LIN {X 98.094,Y 103.990,Z 85.740,A 180.000,B 0.000,C 180.000} C_DIS
LIN {X 98.166,Y 103.986,Z 85.738,A 180.000,B 0.000,C 180.000} C_DIS
LIN {X 98.239,Y 103.980,Z 85.735,A 180.000,B 0.000,C 180.000} C_DIS
LIN {X 98.312,Y 103.973,Z 85.733,A 180.000,B 0.000,C 180.000} C_DIS
LIN {X 98.387,Y 103.963,Z 85.730,A 180.000,B 0.000,C 180.000} C_DIS
LIN {X 98.462,Y 103.954,Z 85.727,A 180.000,B 0.000,C 180.000} C_DIS
LIN {X 98.537,Y 103.942,Z 85.725,A 180.000,B 0.000,C 180.000} C_DIS
LIN {X 98.612,Y 103.930,Z 85.722,A 180.000,B 0.000,C 180.000} C_DIS
LIN {X 98.763,Y 103.903,Z 85.717,A 180.000,B 0.000,C 180.000} C_DIS
LIN {X 98.839,Y 103.890,Z 85.714,A 180.000,B 0.000,C 180.000} C_DIS
LIN {X 98.915,Y 103.876,Z 85.711,A 180.000,B 0.000,C 180.000} C_DIS
LIN {X 98.986,Y 103.863,Z 85.709,A 180.000,B 0.000,C 180.000} C_DIS
LIN {X 99.057,Y 103.847,Z 85.706,A 180.000,B 0.000,C 180.000} C_DIS
LIN {X 99.128,Y 103.830,Z 85.704,A 180.000,B 0.000,C 180.000} C_DIS
LIN {X 99.199,Y 103.813,Z 85.701,A 180.000,B 0.000,C 180.000} C_DIS
LIN {X 99.271,Y 103.794,Z 85.699,A 180.000,B 0.000,C 180.000} C_DIS
LIN {X 99.343,Y 103.773,Z 85.696,A 180.000,B 0.000,C 180.000} C_DIS
LIN {X 99.415,Y 103.751,Z 85.693,A 180.000,B 0.000,C 180.000} C_DIS
LIN {X 99.487,Y 103.729,Z 85.691,A 180.000,B 0.000,C 180.000} C_DIS
LIN {X 99.634,Y 103.684,Z 85.685,A 180.000,B 0.000,C 180.000} C_DIS
LIN {X 99.708,Y 103.661,Z 85.683,A 180.000,B 0.000,C 180.000} C_DIS
LIN {X 99.781,Y 103.637,Z 85.680,A 180.000,B 0.000,C 180.000} C_DIS
LIN {X 99.849,Y 103.613,Z 85.677,A 180.000,B 0.000,C 180.000} C_DIS
LIN {X 99.917,Y 103.588,Z 85.675,A 180.000,B 0.000,C 180.000} C_DIS
LIN {X 99.985,Y 103.562,Z 85.672,A 180.000,B 0.000,C 180.000} C_DIS
LIN {X 100.052,Y 103.534,Z 85.670,A 180.000,B 0.000,C 180.000} C_DIS
LIN {X 100.122,Y 103.504,Z 85.667,A 180.000,B 0.000,C 180.000} C_DIS
LIN {X 100.193,Y 103.473,Z 85.665,A 180.000,B 0.000,C 180.000} C_DIS
LIN {X 100.402,Y 103.379,Z 85.657,A 180.000,B 0.000,C 180.000} C_DIS
LIN {X 100.471,Y 103.347,Z 85.654,A 180.000,B 0.000,C 180.000} C_DIS
LIN {X 100.539,Y 103.314,Z 85.651,A 180.000,B 0.000,C 180.000} C_DIS
LIN {X 100.607,Y 103.280,Z 85.649,A 180.000,B 0.000,C 180.000} C_DIS
LIN {X 100.672,Y 103.247,Z 85.646,A 180.000,B 0.000,C 180.000} C_DIS
LIN {X 100.735,Y 103.212,Z 85.643,A 180.000,B 0.000,C 180.000} C_DIS
LIN {X 100.799,Y 103.176,Z 85.641,A 180.000,B 0.000,C 180.000} C_DIS
LIN {X 100.862,Y 103.139,Z 85.638,A 180.000,B 0.000,C 180.000} C_DIS
LIN {X 100.929,Y 103.099,Z 85.636,A 180.000,B 0.000,C 180.000} C_DIS
LIN {X 101.127,Y 102.977,Z 85.628,A 180.000,B 0.000,C 180.000} C_DIS
LIN {X 101.190,Y 102.938,Z 85.625,A 180.000,B 0.000,C 180.000} C_DIS
LIN {X 101.253,Y 102.897,Z 85.622,A 180.000,B 0.000,C 180.000} C_DIS
LIN {X 101.315,Y 102.856,Z 85.620,A 180.000,B 0.000,C 180.000} C_DIS
LIN {X 101.376,Y 102.813,Z 85.617,A 180.000,B 0.000,C 180.000} C_DIS
LIN {X 101.437,Y 102.769,Z 85.615,A 180.000,B 0.000,C 180.000} C_DIS
LIN {X 101.497,Y 102.725,Z 85.612,A 180.000,B 0.000,C 180.000} C_DIS
LIN {X 101.556,Y 102.680,Z 85.609,A 180.000,B 0.000,C 180.000} C_DIS
LIN {X 101.614,Y 102.633,Z 85.607,A 180.000,B 0.000,C 180.000} C_DIS
LIN {X 101.736,Y 102.536,Z 85.601,A 180.000,B 0.000,C 180.000} C_DIS
LIN {X 101.797,Y 102.487,Z 85.599,A 180.000,B 0.000,C 180.000} C_DIS
LIN {X 101.858,Y 102.437,Z 85.596,A 180.000,B 0.000,C 180.000} C_DIS
LIN {X 101.914,Y 102.391,Z 85.593,A 180.000,B 0.000,C 180.000} C_DIS
LIN {X 101.969,Y 102.343,Z 85.591,A 180.000,B 0.000,C 180.000} C_DIS
LIN {X 102.023,Y 102.293,Z 85.588,A 180.000,B 0.000,C 180.000} C_DIS
LIN {X 102.077,Y 102.244,Z 85.586,A 180.000,B 0.000,C 180.000} C_DIS
LIN {X 102.132,Y 102.191,Z 85.583,A 180.000,B 0.000,C 180.000} C_DIS
LIN {X 102.186,Y 102.137,Z 85.580,A 180.000,B 0.000,C 180.000} C_DIS
LIN {X 102.239,Y 102.082,Z 85.578,A 180.000,B 0.000,C 180.000} C_DIS
LIN {X 102.292,Y 102.027,Z 85.575,A 180.000,B 0.000,C 180.000} C_DIS
LIN {X 102.399,Y 101.917,Z 85.570,A 180.000,B 0.000,C 180.000} C_DIS
LIN {X 102.452,Y 101.862,Z 85.567,A 180.000,B 0.000,C 180.000} C_DIS
LIN {X 102.504,Y 101.806,Z 85.564,A 180.000,B 0.000,C 180.000} C_DIS
LIN {X 102.553,Y 101.749,Z 85.562,A 180.000,B 0.000,C 180.000} C_DIS
LIN {X 102.603,Y 101.692,Z 85.559,A 180.000,B 0.000,C 180.000} C_DIS
LIN {X 102.651,Y 101.635,Z 85.556,A 180.000,B 0.000,C 180.000} C_DIS
LIN {X 102.698,Y 101.575,Z 85.554,A 180.000,B 0.000,C 180.000} C_DIS
LIN {X 102.745,Y 101.515,Z 85.551,A 180.000,B 0.000,C 180.000} C_DIS
LIN {X 102.791,Y 101.455,Z 85.548,A 180.000,B 0.000,C 180.000} C_DIS
LIN {X 102.929,Y 101.272,Z 85.540,A 180.000,B 0.000,C 180.000} C_DIS
LIN {X 102.974,Y 101.211,Z 85.538,A 180.000,B 0.000,C 180.000} C_DIS
LIN {X 103.018,Y 101.148,Z 85.535,A 180.000,B 0.000,C 180.000} C_DIS
LIN {X 103.061,Y 101.085,Z 85.532,A 180.000,B 0.000,C 180.000} C_DIS
LIN {X 103.102,Y 101.024,Z 85.530,A 180.000,B 0.000,C 180.000} C_DIS
LIN {X 103.141,Y 100.961,Z 85.527,A 180.000,B 0.000,C 180.000} C_DIS
LIN {X 103.180,Y 100.898,Z 85.525,A 180.000,B 0.000,C 180.000} C_DIS
LIN {X 103.218,Y 100.835,Z 85.522,A 180.000,B 0.000,C 180.000} C_DIS
LIN {X 103.257,Y 100.767,Z 85.519,A 180.000,B 0.000,C 180.000} C_DIS
LIN {X 103.335,Y 100.632,Z 85.514,A 180.000,B 0.000,C 180.000} C_DIS
LIN {X 103.373,Y 100.564,Z 85.511,A 180.000,B 0.000,C 180.000} C_DIS
LIN {X 103.409,Y 100.498,Z 85.509,A 180.000,B 0.000,C 180.000} C_DIS
LIN {X 103.444,Y 100.433,Z 85.506,A 180.000,B 0.000,C 180.000} C_DIS
LIN {X 103.479,Y 100.367,Z 85.503,A 180.000,B 0.000,C 180.000} C_DIS
LIN {X 103.511,Y 100.300,Z 85.501,A 180.000,B 0.000,C 180.000} C_DIS
LIN {X 103.543,Y 100.231,Z 85.498,A 180.000,B 0.000,C 180.000} C_DIS
LIN {X 103.575,Y 100.162,Z 85.495,A 180.000,B 0.000,C 180.000} C_DIS
LIN {X 103.605,Y 100.093,Z 85.493,A 180.000,B 0.000,C 180.000} C_DIS
LIN {X 103.694,Y 99.878,Z 85.485,A 180.000,B 0.000,C 180.000} C_DIS
LIN {X 103.724,Y 99.806,Z 85.482,A 180.000,B 0.000,C 180.000} C_DIS
LIN {X 103.753,Y 99.734,Z 85.479,A 180.000,B 0.000,C 180.000} C_DIS
LIN {X 103.780,Y 99.664,Z 85.477,A 180.000,B 0.000,C 180.000} C_DIS
LIN {X 103.805,Y 99.594,Z 85.474,A 180.000,B 0.000,C 180.000} C_DIS
LIN {X 103.829,Y 99.524,Z 85.471,A 180.000,B 0.000,C 180.000} C_DIS
LIN {X 103.853,Y 99.453,Z 85.469,A 180.000,B 0.000,C 180.000} C_DIS
LIN {X 103.875,Y 99.380,Z 85.466,A 180.000,B 0.000,C 180.000} C_DIS
LIN {X 103.896,Y 99.306,Z 85.463,A 180.000,B 0.000,C 180.000} C_DIS
LIN {X 103.916,Y 99.232,Z 85.461,A 180.000,B 0.000,C 180.000} C_DIS
LIN {X 103.978,Y 99.008,Z 85.453,A 180.000,B 0.000,C 180.000} C_DIS
LIN {X 103.998,Y 98.933,Z 85.450,A 180.000,B 0.000,C 180.000} C_DIS
LIN {X 104.016,Y 98.858,Z 85.447,A 180.000,B 0.000,C 180.000} C_DIS
LIN {X 104.032,Y 98.785,Z 85.445,A 180.000,B 0.000,C 180.000} C_DIS
LIN {X 104.047,Y 98.712,Z 85.442,A 180.000,B 0.000,C 180.000} C_DIS
LIN {X 104.062,Y 98.639,Z 85.439,A 180.000,B 0.000,C 180.000} C_DIS
LIN {X 104.074,Y 98.565,Z 85.437,A 180.000,B 0.000,C 180.000} C_DIS
LIN {X 104.086,Y 98.489,Z 85.434,A 180.000,B 0.000,C 180.000} C_DIS
LIN {X 104.097,Y 98.412,Z 85.431,A 180.000,B 0.000,C 180.000} C_DIS
LIN {X 104.130,Y 98.183,Z 85.423,A 180.000,B 0.000,C 180.000} C_DIS
LIN {X 104.140,Y 98.107,Z 85.421,A 180.000,B 0.000,C 180.000} C_DIS
LIN {X 104.148,Y 98.032,Z 85.418,A 180.000,B 0.000,C 180.000} C_DIS
LIN {X 104.155,Y 97.956,Z 85.415,A 180.000,B 0.000,C 180.000} C_DIS
LIN {X 104.162,Y 97.880,Z 85.413,A 180.000,B 0.000,C 180.000} C_DIS
LIN {X 104.166,Y 97.803,Z 85.410,A 180.000,B 0.000,C 180.000} C_DIS
LIN {X 104.169,Y 97.727,Z 85.407,A 180.000,B 0.000,C 180.000} C_DIS
LIN {X 104.172,Y 97.651,Z 85.405,A 180.000,B 0.000,C 180.000} C_DIS
LIN {X 104.174,Y 97.573,Z 85.402,A 180.000,B 0.000,C 180.000} C_DIS
LIN {X 104.176,Y 97.419,Z 85.397,A 180.000,B 0.000,C 180.000} C_DIS
LIN {X 104.177,Y 97.342,Z 85.394,A 180.000,B 0.000,C 180.000} C_DIS
LIN {X 104.177,Y 97.266,Z 85.391,A 180.000,B 0.000,C 180.000} C_DIS
LIN {X 104.176,Y 97.191,Z 85.389,A 180.000,B 0.000,C 180.000} C_DIS
LIN {X 104.174,Y 97.115,Z 85.386,A 180.000,B 0.000,C 180.000} C_DIS
LIN {X 104.170,Y 97.039,Z 85.383,A 180.000,B 0.000,C 180.000} C_DIS
LIN {X 104.165,Y 96.963,Z 85.381,A 180.000,B 0.000,C 180.000} C_DIS
LIN {X 104.159,Y 96.886,Z 85.378,A 180.000,B 0.000,C 180.000} C_DIS
LIN {X 104.152,Y 96.810,Z 85.375,A 180.000,B 0.000,C 180.000} C_DIS
LIN {X 104.135,Y 96.656,Z 85.370,A 180.000,B 0.000,C 180.000} C_DIS
LIN {X 104.126,Y 96.578,Z 85.367,A 180.000,B 0.000,C 180.000} C_DIS
LIN {X 104.117,Y 96.500,Z 85.364,A 180.000,B 0.000,C 180.000} C_DIS
LIN {X 104.108,Y 96.423,Z 85.362,A 180.000,B 0.000,C 180.000} C_DIS
LIN {X 104.098,Y 96.348,Z 85.359,A 180.000,B 0.000,C 180.000} C_DIS
LIN {X 104.085,Y 96.273,Z 85.356,A 180.000,B 0.000,C 180.000} C_DIS
LIN {X 104.072,Y 96.199,Z 85.354,A 180.000,B 0.000,C 180.000} C_DIS
LIN {X 104.058,Y 96.124,Z 85.351,A 180.000,B 0.000,C 180.000} C_DIS
LIN {X 104.042,Y 96.049,Z 85.348,A 180.000,B 0.000,C 180.000} C_DIS
LIN {X 104.024,Y 95.973,Z 85.346,A 180.000,B 0.000,C 180.000} C_DIS
LIN {X 103.970,Y 95.747,Z 85.338,A 180.000,B 0.000,C 180.000} C_DIS
LIN {X 103.952,Y 95.672,Z 85.335,A 180.000,B 0.000,C 180.000} C_DIS
LIN {X 103.933,Y 95.596,Z 85.332,A 180.000,B 0.000,C 180.000} C_DIS
LIN {X 103.913,Y 95.521,Z 85.330,A 180.000,B 0.000,C 180.000} C_DIS
LIN {X 103.891,Y 95.449,Z 85.327,A 180.000,B 0.000,C 180.000} C_DIS
LIN {X 103.869,Y 95.376,Z 85.324,A 180.000,B 0.000,C 180.000} C_DIS
LIN {X 103.846,Y 95.304,Z 85.322,A 180.000,B 0.000,C 180.000} C_DIS
LIN {X 103.820,Y 95.233,Z 85.319,A 180.000,B 0.000,C 180.000} C_DIS
LIN {X 103.794,Y 95.160,Z 85.316,A 180.000,B 0.000,C 180.000} C_DIS
LIN {X 103.766,Y 95.087,Z 85.313,A 180.000,B 0.000,C 180.000} C_DIS
LIN {X 103.684,Y 94.869,Z 85.305,A 180.000,B 0.000,C 180.000} C_DIS
LIN {X 103.656,Y 94.797,Z 85.303,A 180.000,B 0.000,C 180.000} C_DIS
LIN {X 103.625,Y 94.726,Z 85.300,A 180.000,B 0.000,C 180.000} C_DIS
LIN {X 103.595,Y 94.655,Z 85.297,A 180.000,B 0.000,C 180.000} C_DIS
LIN {X 103.563,Y 94.585,Z 85.295,A 180.000,B 0.000,C 180.000} C_DIS
LIN {X 103.530,Y 94.516,Z 85.292,A 180.000,B 0.000,C 180.000} C_DIS
LIN {X 103.496,Y 94.448,Z 85.289,A 180.000,B 0.000,C 180.000} C_DIS
LIN {X 103.462,Y 94.380,Z 85.287,A 180.000,B 0.000,C 180.000} C_DIS
LIN {X 103.425,Y 94.311,Z 85.284,A 180.000,B 0.000,C 180.000} C_DIS
LIN {X 103.352,Y 94.172,Z 85.278,A 180.000,B 0.000,C 180.000} C_DIS
LIN {X 103.315,Y 94.103,Z 85.276,A 180.000,B 0.000,C 180.000} C_DIS
LIN {X 103.278,Y 94.037,Z 85.273,A 180.000,B 0.000,C 180.000} C_DIS
LIN {X 103.240,Y 93.970,Z 85.270,A 180.000,B 0.000,C 180.000} C_DIS
LIN {X 103.201,Y 93.904,Z 85.268,A 180.000,B 0.000,C 180.000} C_DIS
LIN {X 103.161,Y 93.840,Z 85.265,A 180.000,B 0.000,C 180.000} C_DIS
LIN {X 103.119,Y 93.775,Z 85.262,A 180.000,B 0.000,C 180.000} C_DIS
LIN {X 103.076,Y 93.710,Z 85.260,A 180.000,B 0.000,C 180.000} C_DIS
LIN {X 103.033,Y 93.646,Z 85.257,A 180.000,B 0.000,C 180.000} C_DIS
LIN {X 102.988,Y 93.583,Z 85.254,A 180.000,B 0.000,C 180.000} C_DIS
LIN {X 102.899,Y 93.455,Z 85.249,A 180.000,B 0.000,C 180.000} C_DIS
LIN {X 102.853,Y 93.392,Z 85.246,A 180.000,B 0.000,C 180.000} C_DIS
LIN {X 102.808,Y 93.329,Z 85.243,A 180.000,B 0.000,C 180.000} C_DIS
LIN {X 102.761,Y 93.267,Z 85.241,A 180.000,B 0.000,C 180.000} C_DIS
LIN {X 102.713,Y 93.206,Z 85.238,A 180.000,B 0.000,C 180.000} C_DIS
LIN {X 102.664,Y 93.146,Z 85.235,A 180.000,B 0.000,C 180.000} C_DIS
LIN {X 102.615,Y 93.087,Z 85.233,A 180.000,B 0.000,C 180.000} C_DIS
LIN {X 102.565,Y 93.028,Z 85.230,A 180.000,B 0.000,C 180.000} C_DIS
LIN {X 102.512,Y 92.970,Z 85.227,A 180.000,B 0.000,C 180.000} C_DIS
LIN {X 102.408,Y 92.856,Z 85.222,A 180.000,B 0.000,C 180.000} C_DIS
LIN {X 102.356,Y 92.798,Z 85.219,A 180.000,B 0.000,C 180.000} C_DIS
LIN {X 102.303,Y 92.741,Z 85.216,A 180.000,B 0.000,C 180.000} C_DIS
LIN {X 102.251,Y 92.684,Z 85.214,A 180.000,B 0.000,C 180.000} C_DIS
LIN {X 102.196,Y 92.629,Z 85.211,A 180.000,B 0.000,C 180.000} C_DIS
LIN {X 102.141,Y 92.575,Z 85.208,A 180.000,B 0.000,C 180.000} C_DIS
LIN {X 102.086,Y 92.521,Z 85.205,A 180.000,B 0.000,C 180.000} C_DIS
LIN {X 102.030,Y 92.469,Z 85.203,A 180.000,B 0.000,C 180.000} C_DIS
LIN {X 101.972,Y 92.418,Z 85.200,A 180.000,B 0.000,C 180.000} C_DIS
LIN {X 101.913,Y 92.366,Z 85.197,A 180.000,B 0.000,C 180.000} C_DIS
LIN {X 101.853,Y 92.315,Z 85.195,A 180.000,B 0.000,C 180.000} C_DIS
LIN {X 101.734,Y 92.213,Z 85.189,A 180.000,B 0.000,C 180.000} C_DIS
LIN {X 101.675,Y 92.162,Z 85.186,A 180.000,B 0.000,C 180.000} C_DIS
LIN {X 101.615,Y 92.113,Z 85.184,A 180.000,B 0.000,C 180.000} C_DIS
LIN {X 101.554,Y 92.066,Z 85.181,A 180.000,B 0.000,C 180.000} C_DIS
LIN {X 101.493,Y 92.018,Z 85.179,A 180.000,B 0.000,C 180.000} C_DIS
LIN {X 101.430,Y 91.972,Z 85.176,A 180.000,B 0.000,C 180.000} C_DIS
LIN {X 101.367,Y 91.927,Z 85.173,A 180.000,B 0.000,C 180.000} C_DIS
LIN {X 101.303,Y 91.883,Z 85.171,A 180.000,B 0.000,C 180.000} C_DIS
LIN {X 101.239,Y 91.839,Z 85.168,A 180.000,B 0.000,C 180.000} C_DIS
LIN {X 101.173,Y 91.796,Z 85.166,A 180.000,B 0.000,C 180.000} C_DIS
LIN {X 101.107,Y 91.753,Z 85.163,A 180.000,B 0.000,C 180.000} C_DIS
LIN {X 101.042,Y 91.710,Z 85.160,A 180.000,B 0.000,C 180.000} C_DIS
LIN {X 100.976,Y 91.667,Z 85.158,A 180.000,B 0.000,C 180.000} C_DIS
LIN {X 100.844,Y 91.587,Z 85.153,A 180.000,B 0.000,C 180.000} C_DIS
LIN {X 100.709,Y 91.510,Z 85.148,A 180.000,B 0.000,C 180.000} C_DIS
LIN {X 100.572,Y 91.437,Z 85.143,A 180.000,B 0.000,C 180.000} C_DIS
LIN {X 100.432,Y 91.368,Z 85.138,A 180.000,B 0.000,C 180.000} C_DIS
LIN {X 100.291,Y 91.299,Z 85.133,A 180.000,B 0.000,C 180.000} C_DIS
LIN {X 100.148,Y 91.233,Z 85.129,A 180.000,B 0.000,C 180.000} C_DIS
LIN {X 100.006,Y 91.171,Z 85.124,A 180.000,B 0.000,C 180.000} C_DIS
LIN {X 99.862,Y 91.114,Z 85.120,A 180.000,B 0.000,C 180.000} C_DIS
LIN {X 99.714,Y 91.062,Z 85.115,A 180.000,B 0.000,C 180.000} C_DIS
LIN {X 99.565,Y 91.012,Z 85.111,A 180.000,B 0.000,C 180.000} C_DIS
LIN {X 99.417,Y 90.962,Z 85.106,A 180.000,B 0.000,C 180.000} C_DIS
LIN {X 99.267,Y 90.916,Z 85.102,A 180.000,B 0.000,C 180.000} C_DIS
LIN {X 99.117,Y 90.875,Z 85.098,A 180.000,B 0.000,C 180.000} C_DIS
LIN {X 98.965,Y 90.840,Z 85.094,A 180.000,B 0.000,C 180.000} C_DIS
LIN {X 98.811,Y 90.808,Z 85.089,A 180.000,B 0.000,C 180.000} C_DIS
LIN {X 98.657,Y 90.777,Z 85.085,A 180.000,B 0.000,C 180.000} C_DIS
LIN {X 98.503,Y 90.748,Z 85.081,A 180.000,B 0.000,C 180.000} C_DIS
LIN {X 98.348,Y 90.724,Z 85.078,A 180.000,B 0.000,C 180.000} C_DIS
LIN {X 98.193,Y 90.706,Z 85.074,A 180.000,B 0.000,C 180.000} C_DIS
LIN {X 98.037,Y 90.692,Z 85.070,A 180.000,B 0.000,C 180.000} C_DIS
LIN {X 97.881,Y 90.680,Z 85.067,A 180.000,B 0.000,C 180.000} C_DIS
LIN {X 97.724,Y 90.670,Z 85.063,A 180.000,B 0.000,C 180.000} C_DIS
LIN {X 97.568,Y 90.663,Z 85.060,A 180.000,B 0.000,C 180.000} C_DIS
LIN {X 97.411,Y 90.662,Z 85.056,A 180.000,B 0.000,C 180.000} C_DIS
LIN {X 97.254,Y 90.666,Z 85.053,A 180.000,B 0.000,C 180.000} C_DIS
LIN {X 97.097,Y 90.674,Z 85.050,A 180.000,B 0.000,C 180.000} C_DIS
LIN {X 96.940,Y 90.682,Z 85.047,A 180.000,B 0.000,C 180.000} C_DIS
LIN {X 96.783,Y 90.694,Z 85.044,A 180.000,B 0.000,C 180.000} C_DIS
LIN {X 96.627,Y 90.710,Z 85.041,A 180.000,B 0.000,C 180.000} C_DIS
LIN {X 96.472,Y 90.731,Z 85.038,A 180.000,B 0.000,C 180.000} C_DIS
LIN {X 96.317,Y 90.758,Z 85.035,A 180.000,B 0.000,C 180.000} C_DIS
LIN {X 96.162,Y 90.786,Z 85.032,A 180.000,B 0.000,C 180.000} C_DIS
LIN {X 96.008,Y 90.815,Z 85.030,A 180.000,B 0.000,C 180.000} C_DIS
LIN {X 95.854,Y 90.849,Z 85.027,A 180.000,B 0.000,C 180.000} C_DIS
LIN {X 95.551,Y 90.931,Z 85.023,A 180.000,B 0.000,C 180.000} C_DIS
LIN {X 95.251,Y 91.026,Z 85.019,A 180.000,B 0.000,C 180.000} C_DIS
LIN {X 94.955,Y 91.132,Z 85.015,A 180.000,B 0.000,C 180.000} C_DIS
LIN {X 94.666,Y 91.257,Z 85.011,A 180.000,B 0.000,C 180.000} C_DIS
LIN {X 94.381,Y 91.390,Z 85.008,A 180.000,B 0.000,C 180.000} C_DIS
LIN {X 94.103,Y 91.538,Z 85.006,A 180.000,B 0.000,C 180.000} C_DIS
LIN {X 93.834,Y 91.702,Z 85.004,A 180.000,B 0.000,C 180.000} C_DIS
LIN {X 93.570,Y 91.873,Z 85.002,A 180.000,B 0.000,C 180.000} C_DIS
LIN {X 93.316,Y 92.059,Z 85.001,A 180.000,B 0.000,C 180.000} C_DIS
LIN {X 93.072,Y 92.259,Z 85.000,A 180.000,B 0.000,C 180.000} C_DIS
LIN {X 92.855,Y 92.446,Z 85.000,A 180.000,B 0.000,C 180.000} C_DIS
; Cutting Move Starts
LIN {X 92.785,Y 92.511,Z 85.000,A 180.000,B 0.000,C 180.000} C_DIS
LIN {X 92.686,Y 92.606,Z 85.000,A 180.000,B 0.000,C 180.000} C_DIS
LIN {X 92.606,Y 92.690,Z 85.000,A 180.000,B 0.000,C 180.000} C_DIS
LIN {X 92.517,Y 92.785,Z 85.000,A 180.000,B 0.000,C 180.000} C_DIS
LIN {X 92.427,Y 92.880,Z 85.000,A 180.000,B 0.000,C 180.000} C_DIS
LIN {X 92.349,Y 92.964,Z 85.000,A 180.000,B 0.000,C 180.000} C_DIS
LIN {X 92.249,Y 93.080,Z 85.000,A 180.000,B 0.000,C 180.000} C_DIS
LIN {X 92.196,Y 93.142,Z 85.000,A 180.000,B 0.000,C 180.000} C_DIS
LIN {X 92.070,Y 93.304,Z 85.000,A 180.000,B 0.000,C 180.000} C_DIS
LIN {X 92.057,Y 93.321,Z 85.000,A 180.000,B 0.000,C 180.000} C_DIS
LIN {X 91.925,Y 93.500,Z 85.000,A 180.000,B 0.000,C 180.000} C_DIS
LIN {X 91.891,Y 93.547,Z 85.000,A 180.000,B 0.000,C 180.000} C_DIS
LIN {X 91.798,Y 93.679,Z 85.000,A 180.000,B 0.000,C 180.000} C_DIS
LIN {X 91.712,Y 93.808,Z 85.000,A 180.000,B 0.000,C 180.000} C_DIS
LIN {X 91.681,Y 93.857,Z 85.000,A 180.000,B 0.000,C 180.000} C_DIS
LIN {X 91.575,Y 94.036,Z 85.000,A 180.000,B 0.000,C 180.000} C_DIS
LIN {X 91.533,Y 94.111,Z 85.000,A 180.000,B 0.000,C 180.000} C_DIS
LIN {X 91.476,Y 94.215,Z 85.000,A 180.000,B 0.000,C 180.000} C_DIS
LIN {X 91.380,Y 94.394,Z 85.000,A 180.000,B 0.000,C 180.000} C_DIS
LIN {X 91.355,Y 94.443,Z 85.000,A 180.000,B 0.000,C 180.000} C_DIS
LIN {X 91.290,Y 94.573,Z 85.000,A 180.000,B 0.000,C 180.000} C_DIS
LIN {X 91.210,Y 94.751,Z 85.000,A 180.000,B 0.000,C 180.000} C_DIS
LIN {X 91.176,Y 94.835,Z 85.000,A 180.000,B 0.000,C 180.000} C_DIS
LIN {X 91.138,Y 94.930,Z 85.000,A 180.000,B 0.000,C 180.000} C_DIS
LIN {X 91.068,Y 95.109,Z 85.000,A 180.000,B 0.000,C 180.000} C_DIS
LIN {X 91.001,Y 95.288,Z 85.000,A 180.000,B 0.000,C 180.000} C_DIS
LIN {X 90.997,Y 95.300,Z 85.000,A 180.000,B 0.000,C 180.000} C_DIS
LIN {X 90.944,Y 95.466,Z 85.000,A 180.000,B 0.000,C 180.000} C_DIS
LIN {X 90.893,Y 95.645,Z 85.000,A 180.000,B 0.000,C 180.000} C_DIS
LIN {X 90.847,Y 95.824,Z 85.000,A 180.000,B 0.000,C 180.000} C_DIS
LIN {X 90.818,Y 95.937,Z 85.000,A 180.000,B 0.000,C 180.000} C_DIS
LIN {X 90.802,Y 96.003,Z 85.000,A 180.000,B 0.000,C 180.000} C_DIS
LIN {X 90.764,Y 96.181,Z 85.000,A 180.000,B 0.000,C 180.000} C_DIS
LIN {X 90.731,Y 96.360,Z 85.000,A 180.000,B 0.000,C 180.000} C_DIS
LIN {X 90.706,Y 96.539,Z 85.000,A 180.000,B 0.000,C 180.000} C_DIS
LIN {X 90.683,Y 96.718,Z 85.000,A 180.000,B 0.000,C 180.000} C_DIS
LIN {X 90.663,Y 96.897,Z 85.000,A 180.000,B 0.000,C 180.000} C_DIS
LIN {X 90.648,Y 97.075,Z 85.000,A 180.000,B 0.000,C 180.000} C_DIS
LIN {X 90.641,Y 97.254,Z 85.000,A 180.000,B 0.000,C 180.000} C_DIS
LIN {X 90.640,Y 97.309,Z 85.000,A 180.000,B 0.000,C 180.000} C_DIS
LIN {X 90.639,Y 97.433,Z 85.000,A 180.000,B 0.000,C 180.000} C_DIS
LIN {X 90.639,Y 97.612,Z 85.000,A 180.000,B 0.000,C 180.000} C_DIS
LIN {X 90.640,Y 97.691,Z 85.000,A 180.000,B 0.000,C 180.000} C_DIS
LIN {X 90.642,Y 97.790,Z 85.000,A 180.000,B 0.000,C 180.000} C_DIS
LIN {X 90.651,Y 97.969,Z 85.000,A 180.000,B 0.000,C 180.000} C_DIS
LIN {X 90.667,Y 98.148,Z 85.000,A 180.000,B 0.000,C 180.000} C_DIS
LIN {X 90.689,Y 98.327,Z 85.000,A 180.000,B 0.000,C 180.000} C_DIS
LIN {X 90.712,Y 98.505,Z 85.000,A 180.000,B 0.000,C 180.000} C_DIS
LIN {X 90.738,Y 98.684,Z 85.000,A 180.000,B 0.000,C 180.000} C_DIS
LIN {X 90.772,Y 98.863,Z 85.000,A 180.000,B 0.000,C 180.000} C_DIS
LIN {X 90.813,Y 99.042,Z 85.000,A 180.000,B 0.000,C 180.000} C_DIS
LIN {X 90.859,Y 99.221,Z 85.000,A 180.000,B 0.000,C 180.000} C_DIS
LIN {X 90.905,Y 99.399,Z 85.000,A 180.000,B 0.000,C 180.000} C_DIS
LIN {X 90.958,Y 99.578,Z 85.000,A 180.000,B 0.000,C 180.000} C_DIS
LIN {X 90.997,Y 99.700,Z 85.000,A 180.000,B 0.000,C 180.000} C_DIS
LIN {X 91.017,Y 99.757,Z 85.000,A 180.000,B 0.000,C 180.000} C_DIS
LIN {X 91.085,Y 99.936,Z 85.000,A 180.000,B 0.000,C 180.000} C_DIS
LIN {X 91.176,Y 100.165,Z 85.000,A 180.000,B 0.000,C 180.000} C_DIS
LIN {X 91.230,Y 100.293,Z 85.000,A 180.000,B 0.000,C 180.000} C_DIS
LIN {X 91.311,Y 100.472,Z 85.000,A 180.000,B 0.000,C 180.000} C_DIS
LIN {X 91.355,Y 100.557,Z 85.000,A 180.000,B 0.000,C 180.000} C_DIS
LIN {X 91.403,Y 100.651,Z 85.000,A 180.000,B 0.000,C 180.000} C_DIS
LIN {X 91.501,Y 100.829,Z 85.000,A 180.000,B 0.000,C 180.000} C_DIS
LIN {X 91.533,Y 100.889,Z 85.000,A 180.000,B 0.000,C 180.000} C_DIS
LIN {X 91.601,Y 101.008,Z 85.000,A 180.000,B 0.000,C 180.000} C_DIS
LIN {X 91.709,Y 101.187,Z 85.000,A 180.000,B 0.000,C 180.000} C_DIS
LIN {X 91.712,Y 101.192,Z 85.000,A 180.000,B 0.000,C 180.000} C_DIS
LIN {X 91.829,Y 101.366,Z 85.000,A 180.000,B 0.000,C 180.000} C_DIS
LIN {X 91.891,Y 101.453,Z 85.000,A 180.000,B 0.000,C 180.000} C_DIS
LIN {X 91.958,Y 101.545,Z 85.000,A 180.000,B 0.000,C 180.000} C_DIS
LIN {X 92.070,Y 101.696,Z 85.000,A 180.000,B 0.000,C 180.000} C_DIS
LIN {X 92.090,Y 101.723,Z 85.000,A 180.000,B 0.000,C 180.000} C_DIS
LIN {X 92.233,Y 101.902,Z 85.000,A 180.000,B 0.000,C 180.000} C_DIS
LIN {X 92.249,Y 101.920,Z 85.000,A 180.000,B 0.000,C 180.000} C_DIS
LIN {X 92.390,Y 102.081,Z 85.000,A 180.000,B 0.000,C 180.000} C_DIS
LIN {X 92.427,Y 102.120,Z 85.000,A 180.000,B 0.000,C 180.000} C_DIS
LIN {X 92.558,Y 102.260,Z 85.000,A 180.000,B 0.000,C 180.000} C_DIS
LIN {X 92.606,Y 102.310,Z 85.000,A 180.000,B 0.000,C 180.000} C_DIS
LIN {X 92.732,Y 102.438,Z 85.000,A 180.000,B 0.000,C 180.000} C_DIS
LIN {X 92.785,Y 102.489,Z 85.000,A 180.000,B 0.000,C 180.000} C_DIS
LIN {X 92.925,Y 102.617,Z 85.000,A 180.000,B 0.000,C 180.000} C_DIS
LIN {X 92.964,Y 102.650,Z 85.000,A 180.000,B 0.000,C 180.000} C_DIS
LIN {X 93.138,Y 102.796,Z 85.000,A 180.000,B 0.000,C 180.000} C_DIS
LIN {X 93.142,Y 102.799,Z 85.000,A 180.000,B 0.000,C 180.000} C_DIS
LIN {X 93.321,Y 102.945,Z 85.000,A 180.000,B 0.000,C 180.000} C_DIS
LIN {X 93.360,Y 102.975,Z 85.000,A 180.000,B 0.000,C 180.000} C_DIS
LIN {X 93.500,Y 103.079,Z 85.000,A 180.000,B 0.000,C 180.000} C_DIS
LIN {X 93.608,Y 103.153,Z 85.000,A 180.000,B 0.000,C 180.000} C_DIS
LIN {X 93.679,Y 103.200,Z 85.000,A 180.000,B 0.000,C 180.000} C_DIS
LIN {X 93.857,Y 103.315,Z 85.000,A 180.000,B 0.000,C 180.000} C_DIS
LIN {X 93.885,Y 103.332,Z 85.000,A 180.000,B 0.000,C 180.000} C_DIS
LIN {X 94.036,Y 103.425,Z 85.000,A 180.000,B 0.000,C 180.000} C_DIS
LIN {X 94.184,Y 103.511,Z 85.000,A 180.000,B 0.000,C 180.000} C_DIS
LIN {X 94.215,Y 103.528,Z 85.000,A 180.000,B 0.000,C 180.000} C_DIS
LIN {X 94.394,Y 103.620,Z 85.000,A 180.000,B 0.000,C 180.000} C_DIS
LIN {X 94.540,Y 103.690,Z 85.000,A 180.000,B 0.000,C 180.000} C_DIS
LIN {X 94.573,Y 103.705,Z 85.000,A 180.000,B 0.000,C 180.000} C_DIS
LIN {X 94.751,Y 103.788,Z 85.000,A 180.000,B 0.000,C 180.000} C_DIS
LIN {X 94.930,Y 103.866,Z 85.000,A 180.000,B 0.000,C 180.000} C_DIS
LIN {X 94.937,Y 103.869,Z 85.000,A 180.000,B 0.000,C 180.000} C_DIS
LIN {X 95.109,Y 103.934,Z 85.000,A 180.000,B 0.000,C 180.000} C_DIS
LIN {X 95.288,Y 103.995,Z 85.000,A 180.000,B 0.000,C 180.000} C_DIS
LIN {X 95.449,Y 104.047,Z 85.000,A 180.000,B 0.000,C 180.000} C_DIS
LIN {X 95.466,Y 104.053,Z 85.000,A 180.000,B 0.000,C 180.000} C_DIS
LIN {X 95.645,Y 104.109,Z 85.000,A 180.000,B 0.000,C 180.000} C_DIS
LIN {X 95.824,Y 104.157,Z 85.000,A 180.000,B 0.000,C 180.000} C_DIS
LIN {X 96.003,Y 104.198,Z 85.000,A 180.000,B 0.000,C 180.000} C_DIS
LIN {X 96.146,Y 104.226,Z 85.000,A 180.000,B 0.000,C 180.000} C_DIS
LIN {X 96.360,Y 104.267,Z 85.000,A 180.000,B 0.000,C 180.000} C_DIS
LIN {X 96.539,Y 104.296,Z 85.000,A 180.000,B 0.000,C 180.000} C_DIS
LIN {X 96.718,Y 104.320,Z 85.000,A 180.000,B 0.000,C 180.000} C_DIS
LIN {X 96.897,Y 104.336,Z 85.000,A 180.000,B 0.000,C 180.000} C_DIS
LIN {X 97.075,Y 104.348,Z 85.000,A 180.000,B 0.000,C 180.000} C_DIS
LIN {X 97.254,Y 104.359,Z 85.000,A 180.000,B 0.000,C 180.000} C_DIS
LIN {X 97.433,Y 104.364,Z 85.000,A 180.000,B 0.000,C 180.000} C_DIS
LIN {X 97.612,Y 104.363,Z 85.000,A 180.000,B 0.000,C 180.000} C_DIS
LIN {X 97.790,Y 104.356,Z 85.000,A 180.000,B 0.000,C 180.000} C_DIS
LIN {X 97.969,Y 104.345,Z 85.000,A 180.000,B 0.000,C 180.000} C_DIS
LIN {X 98.148,Y 104.332,Z 85.000,A 180.000,B 0.000,C 180.000} C_DIS
LIN {X 98.327,Y 104.315,Z 85.000,A 180.000,B 0.000,C 180.000} C_DIS
LIN {X 98.505,Y 104.290,Z 85.000,A 180.000,B 0.000,C 180.000} C_DIS
LIN {X 98.684,Y 104.259,Z 85.000,A 180.000,B 0.000,C 180.000} C_DIS
LIN {X 98.863,Y 104.224,Z 85.000,A 180.000,B 0.000,C 180.000} C_DIS
LIN {X 99.042,Y 104.189,Z 85.000,A 180.000,B 0.000,C 180.000} C_DIS
LIN {X 99.221,Y 104.145,Z 85.000,A 180.000,B 0.000,C 180.000} C_DIS
LIN {X 99.399,Y 104.096,Z 85.000,A 180.000,B 0.000,C 180.000} C_DIS
LIN {X 99.551,Y 104.047,Z 85.000,A 180.000,B 0.000,C 180.000} C_DIS
LIN {X 99.757,Y 103.980,Z 85.000,A 180.000,B 0.000,C 180.000} C_DIS
LIN {X 99.936,Y 103.918,Z 85.000,A 180.000,B 0.000,C 180.000} C_DIS
LIN {X 100.063,Y 103.869,Z 85.000,A 180.000,B 0.000,C 180.000} C_DIS
LIN {X 100.114,Y 103.848,Z 85.000,A 180.000,B 0.000,C 180.000} C_DIS
LIN {X 100.293,Y 103.768,Z 85.000,A 180.000,B 0.000,C 180.000} C_DIS
LIN {X 100.460,Y 103.690,Z 85.000,A 180.000,B 0.000,C 180.000} C_DIS
LIN {X 100.472,Y 103.684,Z 85.000,A 180.000,B 0.000,C 180.000} C_DIS
LIN {X 100.651,Y 103.598,Z 85.000,A 180.000,B 0.000,C 180.000} C_DIS
LIN {X 100.816,Y 103.511,Z 85.000,A 180.000,B 0.000,C 180.000} C_DIS
LIN {X 100.829,Y 103.504,Z 85.000,A 180.000,B 0.000,C 180.000} C_DIS
LIN {X 101.008,Y 103.399,Z 85.000,A 180.000,B 0.000,C 180.000} C_DIS
LIN {X 101.115,Y 103.332,Z 85.000,A 180.000,B 0.000,C 180.000} C_DIS
LIN {X 101.187,Y 103.286,Z 85.000,A 180.000,B 0.000,C 180.000} C_DIS
LIN {X 101.366,Y 103.171,Z 85.000,A 180.000,B 0.000,C 180.000} C_DIS
LIN {X 101.392,Y 103.153,Z 85.000,A 180.000,B 0.000,C 180.000} C_DIS
LIN {X 101.545,Y 103.047,Z 85.000,A 180.000,B 0.000,C 180.000} C_DIS
LIN {X 101.640,Y 102.975,Z 85.000,A 180.000,B 0.000,C 180.000} C_DIS
LIN {X 101.723,Y 102.910,Z 85.000,A 180.000,B 0.000,C 180.000} C_DIS
LIN {X 101.862,Y 102.796,Z 85.000,A 180.000,B 0.000,C 180.000} C_DIS
LIN {X 101.902,Y 102.763,Z 85.000,A 180.000,B 0.000,C 180.000} C_DIS
LIN {X 102.075,Y 102.617,Z 85.000,A 180.000,B 0.000,C 180.000} C_DIS
LIN {X 102.081,Y 102.612,Z 85.000,A 180.000,B 0.000,C 180.000} C_DIS
LIN {X 102.260,Y 102.447,Z 85.000,A 180.000,B 0.000,C 180.000} C_DIS
LIN {X 102.268,Y 102.438,Z 85.000,A 180.000,B 0.000,C 180.000} C_DIS
LIN {X 102.438,Y 102.263,Z 85.000,A 180.000,B 0.000,C 180.000} C_DIS
LIN {X 102.442,Y 102.260,Z 85.000,A 180.000,B 0.000,C 180.000} C_DIS
LIN {X 102.617,Y 102.073,Z 85.000,A 180.000,B 0.000,C 180.000} C_DIS
LIN {X 102.767,Y 101.902,Z 85.000,A 180.000,B 0.000,C 180.000} C_DIS
LIN {X 102.796,Y 101.868,Z 85.000,A 180.000,B 0.000,C 180.000} C_DIS
LIN {X 102.910,Y 101.723,Z 85.000,A 180.000,B 0.000,C 180.000} C_DIS
LIN {X 102.975,Y 101.637,Z 85.000,A 180.000,B 0.000,C 180.000} C_DIS
LIN {X 103.042,Y 101.545,Z 85.000,A 180.000,B 0.000,C 180.000} C_DIS
LIN {X 103.153,Y 101.391,Z 85.000,A 180.000,B 0.000,C 180.000} C_DIS
LIN {X 103.171,Y 101.366,Z 85.000,A 180.000,B 0.000,C 180.000} C_DIS
LIN {X 103.291,Y 101.187,Z 85.000,A 180.000,B 0.000,C 180.000} C_DIS
LIN {X 103.332,Y 101.121,Z 85.000,A 180.000,B 0.000,C 180.000} C_DIS
LIN {X 103.399,Y 101.008,Z 85.000,A 180.000,B 0.000,C 180.000} C_DIS
LIN {X 103.499,Y 100.829,Z 85.000,A 180.000,B 0.000,C 180.000} C_DIS
LIN {X 103.511,Y 100.808,Z 85.000,A 180.000,B 0.000,C 180.000} C_DIS
LIN {X 103.597,Y 100.651,Z 85.000,A 180.000,B 0.000,C 180.000} C_DIS
LIN {X 103.689,Y 100.472,Z 85.000,A 180.000,B 0.000,C 180.000} C_DIS
LIN {X 103.690,Y 100.469,Z 85.000,A 180.000,B 0.000,C 180.000} C_DIS
LIN {X 103.770,Y 100.293,Z 85.000,A 180.000,B 0.000,C 180.000} C_DIS
LIN {X 103.844,Y 100.114,Z 85.000,A 180.000,B 0.000,C 180.000} C_DIS
LIN {X 103.915,Y 99.936,Z 85.000,A 180.000,B 0.000,C 180.000} C_DIS
LIN {X 103.983,Y 99.757,Z 85.000,A 180.000,B 0.000,C 180.000} C_DIS
LIN {X 104.042,Y 99.578,Z 85.000,A 180.000,B 0.000,C 180.000} C_DIS
LIN {X 104.047,Y 99.562,Z 85.000,A 180.000,B 0.000,C 180.000} C_DIS
LIN {X 104.095,Y 99.399,Z 85.000,A 180.000,B 0.000,C 180.000} C_DIS
LIN {X 104.141,Y 99.221,Z 85.000,A 180.000,B 0.000,C 180.000} C_DIS
LIN {X 104.187,Y 99.042,Z 85.000,A 180.000,B 0.000,C 180.000} C_DIS
LIN {X 104.226,Y 98.871,Z 85.000,A 180.000,B 0.000,C 180.000} C_DIS
LIN {X 104.228,Y 98.863,Z 85.000,A 180.000,B 0.000,C 180.000} C_DIS
LIN {X 104.262,Y 98.684,Z 85.000,A 180.000,B 0.000,C 180.000} C_DIS
LIN {X 104.288,Y 98.505,Z 85.000,A 180.000,B 0.000,C 180.000} C_DIS
LIN {X 104.311,Y 98.327,Z 85.000,A 180.000,B 0.000,C 180.000} C_DIS
LIN {X 104.333,Y 98.148,Z 85.000,A 180.000,B 0.000,C 180.000} C_DIS
LIN {X 104.349,Y 97.969,Z 85.000,A 180.000,B 0.000,C 180.000} C_DIS
LIN {X 104.358,Y 97.790,Z 85.000,A 180.000,B 0.000,C 180.000} C_DIS
LIN {X 104.361,Y 97.612,Z 85.000,A 180.000,B 0.000,C 180.000} C_DIS
LIN {X 104.361,Y 97.433,Z 85.000,A 180.000,B 0.000,C 180.000} C_DIS
LIN {X 104.359,Y 97.254,Z 85.000,A 180.000,B 0.000,C 180.000} C_DIS
LIN {X 104.352,Y 97.075,Z 85.000,A 180.000,B 0.000,C 180.000} C_DIS
LIN {X 104.337,Y 96.897,Z 85.000,A 180.000,B 0.000,C 180.000} C_DIS
LIN {X 104.317,Y 96.718,Z 85.000,A 180.000,B 0.000,C 180.000} C_DIS
LIN {X 104.294,Y 96.539,Z 85.000,A 180.000,B 0.000,C 180.000} C_DIS
LIN {X 104.269,Y 96.360,Z 85.000,A 180.000,B 0.000,C 180.000} C_DIS
LIN {X 104.236,Y 96.181,Z 85.000,A 180.000,B 0.000,C 180.000} C_DIS
LIN {X 104.226,Y 96.129,Z 85.000,A 180.000,B 0.000,C 180.000} C_DIS
LIN {X 104.198,Y 96.003,Z 85.000,A 180.000,B 0.000,C 180.000} C_DIS
LIN {X 104.153,Y 95.824,Z 85.000,A 180.000,B 0.000,C 180.000} C_DIS
LIN {X 104.107,Y 95.645,Z 85.000,A 180.000,B 0.000,C 180.000} C_DIS
LIN {X 104.056,Y 95.466,Z 85.000,A 180.000,B 0.000,C 180.000} C_DIS
LIN {X 104.047,Y 95.438,Z 85.000,A 180.000,B 0.000,C 180.000} C_DIS
LIN {X 103.999,Y 95.288,Z 85.000,A 180.000,B 0.000,C 180.000} C_DIS
LIN {X 103.932,Y 95.109,Z 85.000,A 180.000,B 0.000,C 180.000} C_DIS
LIN {X 103.869,Y 94.948,Z 85.000,A 180.000,B 0.000,C 180.000} C_DIS
LIN {X 103.862,Y 94.930,Z 85.000,A 180.000,B 0.000,C 180.000} C_DIS
LIN {X 103.790,Y 94.751,Z 85.000,A 180.000,B 0.000,C 180.000} C_DIS
LIN {X 103.710,Y 94.573,Z 85.000,A 180.000,B 0.000,C 180.000} C_DIS
LIN {X 103.690,Y 94.531,Z 85.000,A 180.000,B 0.000,C 180.000} C_DIS
LIN {X 103.620,Y 94.394,Z 85.000,A 180.000,B 0.000,C 180.000} C_DIS
LIN {X 103.524,Y 94.215,Z 85.000,A 180.000,B 0.000,C 180.000} C_DIS
LIN {X 103.511,Y 94.192,Z 85.000,A 180.000,B 0.000,C 180.000} C_DIS
LIN {X 103.425,Y 94.036,Z 85.000,A 180.000,B 0.000,C 180.000} C_DIS
LIN {X 103.332,Y 93.879,Z 85.000,A 180.000,B 0.000,C 180.000} C_DIS
LIN {X 103.319,Y 93.857,Z 85.000,A 180.000,B 0.000,C 180.000} C_DIS
LIN {X 103.202,Y 93.679,Z 85.000,A 180.000,B 0.000,C 180.000} C_DIS
LIN {X 103.153,Y 93.609,Z 85.000,A 180.000,B 0.000,C 180.000} C_DIS
LIN {X 103.075,Y 93.500,Z 85.000,A 180.000,B 0.000,C 180.000} C_DIS
LIN {X 102.975,Y 93.363,Z 85.000,A 180.000,B 0.000,C 180.000} C_DIS
LIN {X 102.943,Y 93.321,Z 85.000,A 180.000,B 0.000,C 180.000} C_DIS
LIN {X 102.804,Y 93.142,Z 85.000,A 180.000,B 0.000,C 180.000} C_DIS
LIN {X 102.796,Y 93.132,Z 85.000,A 180.000,B 0.000,C 180.000} C_DIS
LIN {X 102.651,Y 92.964,Z 85.000,A 180.000,B 0.000,C 180.000} C_DIS
LIN {X 102.617,Y 92.927,Z 85.000,A 180.000,B 0.000,C 180.000} C_DIS
LIN {X 102.483,Y 92.785,Z 85.000,A 180.000,B 0.000,C 180.000} C_DIS
LIN {X 102.438,Y 92.737,Z 85.000,A 180.000,B 0.000,C 180.000} C_DIS
LIN {X 102.314,Y 92.606,Z 85.000,A 180.000,B 0.000,C 180.000} C_DIS
LIN {X 102.260,Y 92.553,Z 85.000,A 180.000,B 0.000,C 180.000} C_DIS
LIN {X 102.125,Y 92.427,Z 85.000,A 180.000,B 0.000,C 180.000} C_DIS
LIN {X 102.081,Y 92.388,Z 85.000,A 180.000,B 0.000,C 180.000} C_DIS
LIN {X 101.915,Y 92.249,Z 85.000,A 180.000,B 0.000,C 180.000} C_DIS
LIN {X 101.902,Y 92.237,Z 85.000,A 180.000,B 0.000,C 180.000} C_DIS
LIN {X 101.723,Y 92.090,Z 85.000,A 180.000,B 0.000,C 180.000} C_DIS
LIN {X 101.698,Y 92.070,Z 85.000,A 180.000,B 0.000,C 180.000} C_DIS
LIN {X 101.545,Y 91.953,Z 85.000,A 180.000,B 0.000,C 180.000} C_DIS
LIN {X 101.458,Y 91.891,Z 85.000,A 180.000,B 0.000,C 180.000} C_DIS
LIN {X 101.366,Y 91.829,Z 85.000,A 180.000,B 0.000,C 180.000} C_DIS
LIN {X 101.187,Y 91.714,Z 85.000,A 180.000,B 0.000,C 180.000} C_DIS
LIN {X 101.185,Y 91.712,Z 85.000,A 180.000,B 0.000,C 180.000} C_DIS
LIN {X 101.008,Y 91.601,Z 85.000,A 180.000,B 0.000,C 180.000} C_DIS
LIN {X 100.894,Y 91.533,Z 85.000,A 180.000,B 0.000,C 180.000} C_DIS
LIN {X 100.829,Y 91.496,Z 85.000,A 180.000,B 0.000,C 180.000} C_DIS
LIN {X 100.651,Y 91.402,Z 85.000,A 180.000,B 0.000,C 180.000} C_DIS
LIN {X 100.555,Y 91.355,Z 85.000,A 180.000,B 0.000,C 180.000} C_DIS
LIN {X 100.472,Y 91.316,Z 85.000,A 180.000,B 0.000,C 180.000} C_DIS
LIN {X 100.293,Y 91.232,Z 85.000,A 180.000,B 0.000,C 180.000} C_DIS
LIN {X 100.168,Y 91.176,Z 85.000,A 180.000,B 0.000,C 180.000} C_DIS
LIN {X 100.114,Y 91.152,Z 85.000,A 180.000,B 0.000,C 180.000} C_DIS
LIN {X 99.936,Y 91.082,Z 85.000,A 180.000,B 0.000,C 180.000} C_DIS
LIN {X 99.757,Y 91.020,Z 85.000,A 180.000,B 0.000,C 180.000} C_DIS
LIN {X 99.578,Y 90.962,Z 85.000,A 180.000,B 0.000,C 180.000} C_DIS
LIN {X 99.399,Y 90.904,Z 85.000,A 180.000,B 0.000,C 180.000} C_DIS
LIN {X 99.221,Y 90.855,Z 85.000,A 180.000,B 0.000,C 180.000} C_DIS
LIN {X 99.075,Y 90.818,Z 85.000,A 180.000,B 0.000,C 180.000} C_DIS
LIN {X 99.042,Y 90.811,Z 85.000,A 180.000,B 0.000,C 180.000} C_DIS
LIN {X 98.863,Y 90.776,Z 85.000,A 180.000,B 0.000,C 180.000} C_DIS
LIN {X 98.684,Y 90.741,Z 85.000,A 180.000,B 0.000,C 180.000} C_DIS
LIN {X 98.505,Y 90.710,Z 85.000,A 180.000,B 0.000,C 180.000} C_DIS
LIN {X 98.327,Y 90.685,Z 85.000,A 180.000,B 0.000,C 180.000} C_DIS
LIN {X 98.148,Y 90.668,Z 85.000,A 180.000,B 0.000,C 180.000} C_DIS
LIN {X 97.969,Y 90.655,Z 85.000,A 180.000,B 0.000,C 180.000} C_DIS
LIN {X 97.790,Y 90.644,Z 85.000,A 180.000,B 0.000,C 180.000} C_DIS
LIN {X 97.707,Y 90.640,Z 85.000,A 180.000,B 0.000,C 180.000} C_DIS
LIN {X 97.612,Y 90.637,Z 85.000,A 180.000,B 0.000,C 180.000} C_DIS
LIN {X 97.433,Y 90.636,Z 85.000,A 180.000,B 0.000,C 180.000} C_DIS
LIN {X 97.293,Y 90.640,Z 85.000,A 180.000,B 0.000,C 180.000} C_DIS
LIN {X 97.254,Y 90.641,Z 85.000,A 180.000,B 0.000,C 180.000} C_DIS
LIN {X 97.075,Y 90.652,Z 85.000,A 180.000,B 0.000,C 180.000} C_DIS
LIN {X 96.897,Y 90.664,Z 85.000,A 180.000,B 0.000,C 180.000} C_DIS
LIN {X 96.718,Y 90.680,Z 85.000,A 180.000,B 0.000,C 180.000} C_DIS
LIN {X 96.539,Y 90.704,Z 85.000,A 180.000,B 0.000,C 180.000} C_DIS
LIN {X 96.360,Y 90.733,Z 85.000,A 180.000,B 0.000,C 180.000} C_DIS
LIN {X 96.181,Y 90.767,Z 85.000,A 180.000,B 0.000,C 180.000} C_DIS
LIN {X 96.003,Y 90.802,Z 85.000,A 180.000,B 0.000,C 180.000} C_DIS
LIN {X 95.925,Y 90.818,Z 85.000,A 180.000,B 0.000,C 180.000} C_DIS
LIN {X 95.824,Y 90.843,Z 85.000,A 180.000,B 0.000,C 180.000} C_DIS
LIN {X 95.645,Y 90.891,Z 85.000,A 180.000,B 0.000,C 180.000} C_DIS
LIN {X 95.466,Y 90.947,Z 85.000,A 180.000,B 0.000,C 180.000} C_DIS
LIN {X 95.312,Y 90.997,Z 85.000,A 180.000,B 0.000,C 180.000} C_DIS
LIN {X 95.288,Y 91.005,Z 85.000,A 180.000,B 0.000,C 180.000} C_DIS
LIN {X 95.109,Y 91.066,Z 85.000,A 180.000,B 0.000,C 180.000} C_DIS
LIN {X 94.930,Y 91.134,Z 85.000,A 180.000,B 0.000,C 180.000} C_DIS
LIN {X 94.832,Y 91.176,Z 85.000,A 180.000,B 0.000,C 180.000} C_DIS
LIN {X 94.751,Y 91.212,Z 85.000,A 180.000,B 0.000,C 180.000} C_DIS
LIN {X 94.573,Y 91.295,Z 85.000,A 180.000,B 0.000,C 180.000} C_DIS
LIN {X 94.445,Y 91.355,Z 85.000,A 180.000,B 0.000,C 180.000} C_DIS
LIN {X 94.394,Y 91.380,Z 85.000,A 180.000,B 0.000,C 180.000} C_DIS
LIN {X 94.215,Y 91.472,Z 85.000,A 180.000,B 0.000,C 180.000} C_DIS
LIN {X 94.106,Y 91.533,Z 85.000,A 180.000,B 0.000,C 180.000} C_DIS
LIN {X 94.036,Y 91.575,Z 85.000,A 180.000,B 0.000,C 180.000} C_DIS
LIN {X 93.857,Y 91.685,Z 85.000,A 180.000,B 0.000,C 180.000} C_DIS
LIN {X 93.815,Y 91.712,Z 85.000,A 180.000,B 0.000,C 180.000} C_DIS
LIN {X 93.679,Y 91.800,Z 85.000,A 180.000,B 0.000,C 180.000} C_DIS
LIN {X 93.542,Y 91.891,Z 85.000,A 180.000,B 0.000,C 180.000} C_DIS
LIN {X 93.500,Y 91.921,Z 85.000,A 180.000,B 0.000,C 180.000} C_DIS
LIN {X 93.321,Y 92.055,Z 85.000,A 180.000,B 0.000,C 180.000} C_DIS
LIN {X 93.302,Y 92.070,Z 85.000,A 180.000,B 0.000,C 180.000} C_DIS
LIN {X 93.142,Y 92.201,Z 85.000,A 180.000,B 0.000,C 180.000} C_DIS
LIN {X 93.085,Y 92.249,Z 85.000,A 180.000,B 0.000,C 180.000} C_DIS
LIN {X 92.964,Y 92.350,Z 85.000,A 180.000,B 0.000,C 180.000} C_DIS
LIN {X 92.875,Y 92.427,Z 85.000,A 180.000,B 0.000,C 180.000} C_DIS
LIN {X 92.855,Y 92.446,Z 85.000,A 180.000,B 0.000,C 180.000} C_DIS
; Link Move Starts
LIN {X 92.645,Y 92.649,Z 85.000,A 180.000,B 0.000,C 180.000} C_DIS
LIN {X 92.433,Y 92.873,Z 84.999,A 180.000,B 0.000,C 180.000} C_DIS
LIN {X 92.244,Y 93.083,Z 84.998,A 180.000,B 0.000,C 180.000} C_DIS
LIN {X 92.060,Y 93.313,Z 84.997,A 180.000,B 0.000,C 180.000} C_DIS
LIN {X 91.877,Y 93.562,Z 84.995,A 180.000,B 0.000,C 180.000} C_DIS
LIN {X 91.716,Y 93.796,Z 84.992,A 180.000,B 0.000,C 180.000} C_DIS
LIN {X 91.563,Y 94.048,Z 84.990,A 180.000,B 0.000,C 180.000} C_DIS
LIN {X 91.414,Y 94.315,Z 84.987,A 180.000,B 0.000,C 180.000} C_DIS
LIN {X 91.278,Y 94.580,Z 84.983,A 180.000,B 0.000,C 180.000} C_DIS
LIN {X 91.165,Y 94.837,Z 84.979,A 180.000,B 0.000,C 180.000} C_DIS
LIN {X 91.052,Y 95.119,Z 84.975,A 180.000,B 0.000,C 180.000} C_DIS
LIN {X 90.952,Y 95.396,Z 84.971,A 180.000,B 0.000,C 180.000} C_DIS
LIN {X 90.870,Y 95.671,Z 84.966,A 180.000,B 0.000,C 180.000} C_DIS
LIN {X 90.831,Y 95.818,Z 84.963,A 180.000,B 0.000,C 180.000} C_DIS
LIN {X 90.792,Y 95.966,Z 84.960,A 180.000,B 0.000,C 180.000} C_DIS
LIN {X 90.757,Y 96.112,Z 84.958,A 180.000,B 0.000,C 180.000} C_DIS
LIN {X 90.727,Y 96.258,Z 84.955,A 180.000,B 0.000,C 180.000} C_DIS
LIN {X 90.703,Y 96.400,Z 84.952,A 180.000,B 0.000,C 180.000} C_DIS
LIN {X 90.681,Y 96.543,Z 84.949,A 180.000,B 0.000,C 180.000} C_DIS
LIN {X 90.661,Y 96.691,Z 84.946,A 180.000,B 0.000,C 180.000} C_DIS
LIN {X 90.641,Y 96.840,Z 84.943,A 180.000,B 0.000,C 180.000} C_DIS
LIN {X 90.627,Y 96.982,Z 84.939,A 180.000,B 0.000,C 180.000} C_DIS
LIN {X 90.615,Y 97.124,Z 84.936,A 180.000,B 0.000,C 180.000} C_DIS
LIN {X 90.609,Y 97.277,Z 84.933,A 180.000,B 0.000,C 180.000} C_DIS
LIN {X 90.606,Y 97.431,Z 84.929,A 180.000,B 0.000,C 180.000} C_DIS
LIN {X 90.604,Y 97.580,Z 84.926,A 180.000,B 0.000,C 180.000} C_DIS
LIN {X 90.604,Y 97.730,Z 84.922,A 180.000,B 0.000,C 180.000} C_DIS
LIN {X 90.607,Y 97.874,Z 84.918,A 180.000,B 0.000,C 180.000} C_DIS
LIN {X 90.616,Y 98.018,Z 84.915,A 180.000,B 0.000,C 180.000} C_DIS
LIN {X 90.627,Y 98.166,Z 84.911,A 180.000,B 0.000,C 180.000} C_DIS
LIN {X 90.643,Y 98.314,Z 84.907,A 180.000,B 0.000,C 180.000} C_DIS
LIN {X 90.661,Y 98.468,Z 84.903,A 180.000,B 0.000,C 180.000} C_DIS
LIN {X 90.680,Y 98.621,Z 84.898,A 180.000,B 0.000,C 180.000} C_DIS
LIN {X 90.703,Y 98.764,Z 84.894,A 180.000,B 0.000,C 180.000} C_DIS
LIN {X 90.729,Y 98.907,Z 84.890,A 180.000,B 0.000,C 180.000} C_DIS
LIN {X 90.760,Y 99.050,Z 84.886,A 180.000,B 0.000,C 180.000} C_DIS
LIN {X 90.795,Y 99.193,Z 84.882,A 180.000,B 0.000,C 180.000} C_DIS
LIN {X 90.830,Y 99.336,Z 84.877,A 180.000,B 0.000,C 180.000} C_DIS
LIN {X 90.865,Y 99.479,Z 84.873,A 180.000,B 0.000,C 180.000} C_DIS
LIN {X 90.909,Y 99.625,Z 84.868,A 180.000,B 0.000,C 180.000} C_DIS
LIN {X 90.955,Y 99.771,Z 84.864,A 180.000,B 0.000,C 180.000} C_DIS
LIN {X 91.005,Y 99.909,Z 84.859,A 180.000,B 0.000,C 180.000} C_DIS
LIN {X 91.056,Y 100.047,Z 84.854,A 180.000,B 0.000,C 180.000} C_DIS
LIN {X 91.109,Y 100.186,Z 84.850,A 180.000,B 0.000,C 180.000} C_DIS
LIN {X 91.165,Y 100.324,Z 84.845,A 180.000,B 0.000,C 180.000} C_DIS
LIN {X 91.223,Y 100.460,Z 84.840,A 180.000,B 0.000,C 180.000} C_DIS
LIN {X 91.287,Y 100.594,Z 84.835,A 180.000,B 0.000,C 180.000} C_DIS
LIN {X 91.321,Y 100.661,Z 84.833,A 180.000,B 0.000,C 180.000} C_DIS
LIN {X 91.355,Y 100.728,Z 84.830,A 180.000,B 0.000,C 180.000} C_DIS
LIN {X 91.390,Y 100.795,Z 84.828,A 180.000,B 0.000,C 180.000} C_DIS
LIN {X 91.461,Y 100.929,Z 84.822,A 180.000,B 0.000,C 180.000} C_DIS
LIN {X 91.497,Y 100.996,Z 84.820,A 180.000,B 0.000,C 180.000} C_DIS
LIN {X 91.534,Y 101.062,Z 84.817,A 180.000,B 0.000,C 180.000} C_DIS
LIN {X 91.572,Y 101.128,Z 84.815,A 180.000,B 0.000,C 180.000} C_DIS
LIN {X 91.645,Y 101.252,Z 84.810,A 180.000,B 0.000,C 180.000} C_DIS
LIN {X 91.684,Y 101.312,Z 84.807,A 180.000,B 0.000,C 180.000} C_DIS
LIN {X 91.723,Y 101.372,Z 84.805,A 180.000,B 0.000,C 180.000} C_DIS
LIN {X 91.765,Y 101.436,Z 84.802,A 180.000,B 0.000,C 180.000} C_DIS
LIN {X 91.809,Y 101.499,Z 84.799,A 180.000,B 0.000,C 180.000} C_DIS
LIN {X 91.897,Y 101.625,Z 84.794,A 180.000,B 0.000,C 180.000} C_DIS
LIN {X 91.939,Y 101.684,Z 84.791,A 180.000,B 0.000,C 180.000} C_DIS
LIN {X 91.982,Y 101.744,Z 84.789,A 180.000,B 0.000,C 180.000} C_DIS
LIN {X 92.025,Y 101.803,Z 84.786,A 180.000,B 0.000,C 180.000} C_DIS
LIN {X 92.068,Y 101.861,Z 84.784,A 180.000,B 0.000,C 180.000} C_DIS
LIN {X 92.115,Y 101.920,Z 84.781,A 180.000,B 0.000,C 180.000} C_DIS
LIN {X 92.162,Y 101.978,Z 84.778,A 180.000,B 0.000,C 180.000} C_DIS
LIN {X 92.210,Y 102.037,Z 84.776,A 180.000,B 0.000,C 180.000} C_DIS
LIN {X 92.258,Y 102.094,Z 84.773,A 180.000,B 0.000,C 180.000} C_DIS
LIN {X 92.310,Y 102.151,Z 84.770,A 180.000,B 0.000,C 180.000} C_DIS
LIN {X 92.413,Y 102.265,Z 84.765,A 180.000,B 0.000,C 180.000} C_DIS
LIN {X 92.464,Y 102.321,Z 84.762,A 180.000,B 0.000,C 180.000} C_DIS
LIN {X 92.566,Y 102.433,Z 84.757,A 180.000,B 0.000,C 180.000} C_DIS
LIN {X 92.618,Y 102.487,Z 84.755,A 180.000,B 0.000,C 180.000} C_DIS
LIN {X 92.672,Y 102.541,Z 84.752,A 180.000,B 0.000,C 180.000} C_DIS
LIN {X 92.723,Y 102.591,Z 84.749,A 180.000,B 0.000,C 180.000} C_DIS
LIN {X 92.775,Y 102.641,Z 84.747,A 180.000,B 0.000,C 180.000} C_DIS
LIN {X 92.827,Y 102.690,Z 84.744,A 180.000,B 0.000,C 180.000} C_DIS
LIN {X 92.881,Y 102.738,Z 84.742,A 180.000,B 0.000,C 180.000} C_DIS
LIN {X 92.940,Y 102.789,Z 84.739,A 180.000,B 0.000,C 180.000} C_DIS
LIN {X 92.999,Y 102.840,Z 84.736,A 180.000,B 0.000,C 180.000} C_DIS
LIN {X 93.173,Y 102.989,Z 84.728,A 180.000,B 0.000,C 180.000} C_DIS
LIN {X 93.229,Y 103.036,Z 84.726,A 180.000,B 0.000,C 180.000} C_DIS
LIN {X 93.287,Y 103.081,Z 84.723,A 180.000,B 0.000,C 180.000} C_DIS
LIN {X 93.344,Y 103.126,Z 84.721,A 180.000,B 0.000,C 180.000} C_DIS
LIN {X 93.404,Y 103.172,Z 84.718,A 180.000,B 0.000,C 180.000} C_DIS
LIN {X 93.465,Y 103.217,Z 84.715,A 180.000,B 0.000,C 180.000} C_DIS
LIN {X 93.527,Y 103.260,Z 84.713,A 180.000,B 0.000,C 180.000} C_DIS
LIN {X 93.589,Y 103.303,Z 84.710,A 180.000,B 0.000,C 180.000} C_DIS
LIN {X 93.653,Y 103.346,Z 84.707,A 180.000,B 0.000,C 180.000} C_DIS
LIN {X 93.782,Y 103.431,Z 84.702,A 180.000,B 0.000,C 180.000} C_DIS
LIN {X 93.846,Y 103.474,Z 84.699,A 180.000,B 0.000,C 180.000} C_DIS
LIN {X 93.908,Y 103.514,Z 84.697,A 180.000,B 0.000,C 180.000} C_DIS
LIN {X 93.971,Y 103.553,Z 84.694,A 180.000,B 0.000,C 180.000} C_DIS
LIN {X 94.035,Y 103.591,Z 84.692,A 180.000,B 0.000,C 180.000} C_DIS
LIN {X 94.098,Y 103.629,Z 84.689,A 180.000,B 0.000,C 180.000} C_DIS
LIN {X 94.162,Y 103.665,Z 84.686,A 180.000,B 0.000,C 180.000} C_DIS
LIN {X 94.227,Y 103.700,Z 84.684,A 180.000,B 0.000,C 180.000} C_DIS
LIN {X 94.292,Y 103.735,Z 84.681,A 180.000,B 0.000,C 180.000} C_DIS
LIN {X 94.357,Y 103.769,Z 84.679,A 180.000,B 0.000,C 180.000} C_DIS
LIN {X 94.427,Y 103.804,Z 84.676,A 180.000,B 0.000,C 180.000} C_DIS
LIN {X 94.567,Y 103.872,Z 84.671,A 180.000,B 0.000,C 180.000} C_DIS
LIN {X 94.637,Y 103.906,Z 84.668,A 180.000,B 0.000,C 180.000} C_DIS
LIN {X 94.704,Y 103.938,Z 84.665,A 180.000,B 0.000,C 180.000} C_DIS
LIN {X 94.770,Y 103.969,Z 84.663,A 180.000,B 0.000,C 180.000} C_DIS
LIN {X 94.838,Y 103.999,Z 84.660,A 180.000,B 0.000,C 180.000} C_DIS
LIN {X 94.906,Y 104.028,Z 84.658,A 180.000,B 0.000,C 180.000} C_DIS
LIN {X 95.045,Y 104.083,Z 84.652,A 180.000,B 0.000,C 180.000} C_DIS
LIN {X 95.115,Y 104.110,Z 84.650,A 180.000,B 0.000,C 180.000} C_DIS
LIN {X 95.186,Y 104.135,Z 84.647,A 180.000,B 0.000,C 180.000} C_DIS
LIN {X 95.334,Y 104.186,Z 84.642,A 180.000,B 0.000,C 180.000} C_DIS
LIN {X 95.408,Y 104.211,Z 84.639,A 180.000,B 0.000,C 180.000} C_DIS
LIN {X 95.482,Y 104.236,Z 84.636,A 180.000,B 0.000,C 180.000} C_DIS
LIN {X 95.552,Y 104.260,Z 84.634,A 180.000,B 0.000,C 180.000} C_DIS
LIN {X 95.623,Y 104.282,Z 84.631,A 180.000,B 0.000,C 180.000} C_DIS
LIN {X 95.694,Y 104.302,Z 84.628,A 180.000,B 0.000,C 180.000} C_DIS
LIN {X 95.766,Y 104.322,Z 84.626,A 180.000,B 0.000,C 180.000} C_DIS
LIN {X 95.838,Y 104.342,Z 84.623,A 180.000,B 0.000,C 180.000} C_DIS
LIN {X 95.911,Y 104.360,Z 84.621,A 180.000,B 0.000,C 180.000} C_DIS
LIN {X 95.985,Y 104.376,Z 84.618,A 180.000,B 0.000,C 180.000} C_DIS
LIN {X 96.058,Y 104.392,Z 84.615,A 180.000,B 0.000,C 180.000} C_DIS
LIN {X 96.134,Y 104.408,Z 84.613,A 180.000,B 0.000,C 180.000} C_DIS
LIN {X 96.287,Y 104.440,Z 84.607,A 180.000,B 0.000,C 180.000} C_DIS
LIN {X 96.363,Y 104.455,Z 84.604,A 180.000,B 0.000,C 180.000} C_DIS
LIN {X 96.436,Y 104.469,Z 84.602,A 180.000,B 0.000,C 180.000} C_DIS
LIN {X 96.509,Y 104.481,Z 84.599,A 180.000,B 0.000,C 180.000} C_DIS
LIN {X 96.583,Y 104.493,Z 84.597,A 180.000,B 0.000,C 180.000} C_DIS
LIN {X 96.656,Y 104.504,Z 84.594,A 180.000,B 0.000,C 180.000} C_DIS
LIN {X 96.731,Y 104.513,Z 84.591,A 180.000,B 0.000,C 180.000} C_DIS
LIN {X 96.805,Y 104.521,Z 84.589,A 180.000,B 0.000,C 180.000} C_DIS
LIN {X 96.880,Y 104.528,Z 84.586,A 180.000,B 0.000,C 180.000} C_DIS
LIN {X 96.954,Y 104.535,Z 84.584,A 180.000,B 0.000,C 180.000} C_DIS
LIN {X 97.187,Y 104.553,Z 84.575,A 180.000,B 0.000,C 180.000} C_DIS
LIN {X 97.264,Y 104.559,Z 84.573,A 180.000,B 0.000,C 180.000} C_DIS
LIN {X 97.339,Y 104.562,Z 84.570,A 180.000,B 0.000,C 180.000} C_DIS
LIN {X 97.414,Y 104.565,Z 84.568,A 180.000,B 0.000,C 180.000} C_DIS
LIN {X 97.489,Y 104.568,Z 84.565,A 180.000,B 0.000,C 180.000} C_DIS
LIN {X 97.564,Y 104.569,Z 84.562,A 180.000,B 0.000,C 180.000} C_DIS
LIN {X 97.715,Y 104.567,Z 84.557,A 180.000,B 0.000,C 180.000} C_DIS
LIN {X 97.790,Y 104.565,Z 84.554,A 180.000,B 0.000,C 180.000} C_DIS
LIN {X 97.865,Y 104.561,Z 84.552,A 180.000,B 0.000,C 180.000} C_DIS
LIN {X 98.019,Y 104.554,Z 84.546,A 180.000,B 0.000,C 180.000} C_DIS
LIN {X 98.096,Y 104.550,Z 84.544,A 180.000,B 0.000,C 180.000} C_DIS
LIN {X 98.248,Y 104.540,Z 84.538,A 180.000,B 0.000,C 180.000} C_DIS
LIN {X 98.322,Y 104.534,Z 84.536,A 180.000,B 0.000,C 180.000} C_DIS
LIN {X 98.396,Y 104.525,Z 84.533,A 180.000,B 0.000,C 180.000} C_DIS
LIN {X 98.471,Y 104.516,Z 84.531,A 180.000,B 0.000,C 180.000} C_DIS
LIN {X 98.546,Y 104.507,Z 84.528,A 180.000,B 0.000,C 180.000} C_DIS
LIN {X 98.622,Y 104.496,Z 84.525,A 180.000,B 0.000,C 180.000} C_DIS
LIN {X 98.698,Y 104.483,Z 84.523,A 180.000,B 0.000,C 180.000} C_DIS
LIN {X 98.849,Y 104.456,Z 84.517,A 180.000,B 0.000,C 180.000} C_DIS
LIN {X 98.926,Y 104.443,Z 84.514,A 180.000,B 0.000,C 180.000} C_DIS
LIN {X 99.002,Y 104.429,Z 84.512,A 180.000,B 0.000,C 180.000} C_DIS
LIN {X 99.078,Y 104.415,Z 84.509,A 180.000,B 0.000,C 180.000} C_DIS
LIN {X 99.151,Y 104.400,Z 84.506,A 180.000,B 0.000,C 180.000} C_DIS
LIN {X 99.223,Y 104.383,Z 84.504,A 180.000,B 0.000,C 180.000} C_DIS
LIN {X 99.296,Y 104.366,Z 84.501,A 180.000,B 0.000,C 180.000} C_DIS
LIN {X 99.368,Y 104.348,Z 84.499,A 180.000,B 0.000,C 180.000} C_DIS
LIN {X 99.443,Y 104.328,Z 84.496,A 180.000,B 0.000,C 180.000} C_DIS
LIN {X 99.517,Y 104.306,Z 84.493,A 180.000,B 0.000,C 180.000} C_DIS
LIN {X 99.591,Y 104.284,Z 84.491,A 180.000,B 0.000,C 180.000} C_DIS
LIN {X 99.665,Y 104.261,Z 84.488,A 180.000,B 0.000,C 180.000} C_DIS
LIN {X 99.811,Y 104.217,Z 84.483,A 180.000,B 0.000,C 180.000} C_DIS
LIN {X 99.884,Y 104.194,Z 84.480,A 180.000,B 0.000,C 180.000} C_DIS
LIN {X 99.957,Y 104.170,Z 84.477,A 180.000,B 0.000,C 180.000} C_DIS
LIN {X 100.027,Y 104.145,Z 84.475,A 180.000,B 0.000,C 180.000} C_DIS
LIN {X 100.098,Y 104.119,Z 84.472,A 180.000,B 0.000,C 180.000} C_DIS
LIN {X 100.169,Y 104.093,Z 84.469,A 180.000,B 0.000,C 180.000} C_DIS
LIN {X 100.238,Y 104.065,Z 84.467,A 180.000,B 0.000,C 180.000} C_DIS
LIN {X 100.310,Y 104.034,Z 84.464,A 180.000,B 0.000,C 180.000} C_DIS
LIN {X 100.381,Y 104.004,Z 84.461,A 180.000,B 0.000,C 180.000} C_DIS
LIN {X 100.453,Y 103.973,Z 84.459,A 180.000,B 0.000,C 180.000} C_DIS
LIN {X 100.663,Y 103.878,Z 84.450,A 180.000,B 0.000,C 180.000} C_DIS
LIN {X 100.732,Y 103.845,Z 84.448,A 180.000,B 0.000,C 180.000} C_DIS
LIN {X 100.801,Y 103.811,Z 84.445,A 180.000,B 0.000,C 180.000} C_DIS
LIN {X 100.869,Y 103.778,Z 84.442,A 180.000,B 0.000,C 180.000} C_DIS
LIN {X 100.937,Y 103.743,Z 84.440,A 180.000,B 0.000,C 180.000} C_DIS
LIN {X 101.003,Y 103.707,Z 84.437,A 180.000,B 0.000,C 180.000} C_DIS
LIN {X 101.136,Y 103.631,Z 84.432,A 180.000,B 0.000,C 180.000} C_DIS
LIN {X 101.203,Y 103.592,Z 84.429,A 180.000,B 0.000,C 180.000} C_DIS
LIN {X 101.400,Y 103.471,Z 84.421,A 180.000,B 0.000,C 180.000} C_DIS
LIN {X 101.466,Y 103.430,Z 84.418,A 180.000,B 0.000,C 180.000} C_DIS
LIN {X 101.596,Y 103.346,Z 84.413,A 180.000,B 0.000,C 180.000} C_DIS
LIN {X 101.658,Y 103.304,Z 84.410,A 180.000,B 0.000,C 180.000} C_DIS
LIN {X 101.719,Y 103.261,Z 84.408,A 180.000,B 0.000,C 180.000} C_DIS
LIN {X 101.780,Y 103.217,Z 84.405,A 180.000,B 0.000,C 180.000} C_DIS
LIN {X 101.840,Y 103.173,Z 84.402,A 180.000,B 0.000,C 180.000} C_DIS
LIN {X 101.902,Y 103.126,Z 84.400,A 180.000,B 0.000,C 180.000} C_DIS
LIN {X 101.963,Y 103.077,Z 84.397,A 180.000,B 0.000,C 180.000} C_DIS
LIN {X 102.085,Y 102.980,Z 84.392,A 180.000,B 0.000,C 180.000} C_DIS
LIN {X 102.144,Y 102.932,Z 84.389,A 180.000,B 0.000,C 180.000} C_DIS
LIN {X 102.203,Y 102.883,Z 84.386,A 180.000,B 0.000,C 180.000} C_DIS
LIN {X 102.263,Y 102.835,Z 84.384,A 180.000,B 0.000,C 180.000} C_DIS
LIN {X 102.321,Y 102.785,Z 84.381,A 180.000,B 0.000,C 180.000} C_DIS
LIN {X 102.377,Y 102.734,Z 84.378,A 180.000,B 0.000,C 180.000} C_DIS
LIN {X 102.434,Y 102.683,Z 84.376,A 180.000,B 0.000,C 180.000} C_DIS
LIN {X 102.490,Y 102.631,Z 84.373,A 180.000,B 0.000,C 180.000} C_DIS
LIN {X 102.545,Y 102.578,Z 84.370,A 180.000,B 0.000,C 180.000} C_DIS
LIN {X 102.599,Y 102.522,Z 84.368,A 180.000,B 0.000,C 180.000} C_DIS
LIN {X 102.654,Y 102.466,Z 84.365,A 180.000,B 0.000,C 180.000} C_DIS
LIN {X 102.708,Y 102.410,Z 84.362,A 180.000,B 0.000,C 180.000} C_DIS
LIN {X 102.816,Y 102.299,Z 84.357,A 180.000,B 0.000,C 180.000} C_DIS
LIN {X 102.869,Y 102.244,Z 84.354,A 180.000,B 0.000,C 180.000} C_DIS
LIN {X 102.921,Y 102.188,Z 84.351,A 180.000,B 0.000,C 180.000} C_DIS
LIN {X 102.972,Y 102.130,Z 84.349,A 180.000,B 0.000,C 180.000} C_DIS
LIN {X 103.022,Y 102.072,Z 84.346,A 180.000,B 0.000,C 180.000} C_DIS
LIN {X 103.072,Y 102.014,Z 84.343,A 180.000,B 0.000,C 180.000} C_DIS
LIN {X 103.120,Y 101.955,Z 84.341,A 180.000,B 0.000,C 180.000} C_DIS
LIN {X 103.168,Y 101.894,Z 84.338,A 180.000,B 0.000,C 180.000} C_DIS
LIN {X 103.215,Y 101.833,Z 84.335,A 180.000,B 0.000,C 180.000} C_DIS
LIN {X 103.263,Y 101.771,Z 84.332,A 180.000,B 0.000,C 180.000} C_DIS
LIN {X 103.357,Y 101.646,Z 84.327,A 180.000,B 0.000,C 180.000} C_DIS
LIN {X 103.403,Y 101.584,Z 84.324,A 180.000,B 0.000,C 180.000} C_DIS
LIN {X 103.448,Y 101.522,Z 84.322,A 180.000,B 0.000,C 180.000} C_DIS
LIN {X 103.492,Y 101.458,Z 84.319,A 180.000,B 0.000,C 180.000} C_DIS
LIN {X 103.536,Y 101.395,Z 84.316,A 180.000,B 0.000,C 180.000} C_DIS
LIN {X 103.579,Y 101.331,Z 84.314,A 180.000,B 0.000,C 180.000} C_DIS
LIN {X 103.620,Y 101.266,Z 84.311,A 180.000,B 0.000,C 180.000} C_DIS
LIN {X 103.700,Y 101.135,Z 84.306,A 180.000,B 0.000,C 180.000} C_DIS
LIN {X 103.739,Y 101.068,Z 84.303,A 180.000,B 0.000,C 180.000} C_DIS
LIN {X 103.816,Y 100.934,Z 84.297,A 180.000,B 0.000,C 180.000} C_DIS
LIN {X 103.854,Y 100.867,Z 84.295,A 180.000,B 0.000,C 180.000} C_DIS
LIN {X 103.892,Y 100.799,Z 84.292,A 180.000,B 0.000,C 180.000} C_DIS
LIN {X 103.928,Y 100.731,Z 84.289,A 180.000,B 0.000,C 180.000} C_DIS
LIN {X 103.965,Y 100.663,Z 84.287,A 180.000,B 0.000,C 180.000} C_DIS
LIN {X 104.000,Y 100.594,Z 84.284,A 180.000,B 0.000,C 180.000} C_DIS
LIN {X 104.033,Y 100.525,Z 84.281,A 180.000,B 0.000,C 180.000} C_DIS
LIN {X 104.066,Y 100.456,Z 84.279,A 180.000,B 0.000,C 180.000} C_DIS
LIN {X 104.098,Y 100.386,Z 84.276,A 180.000,B 0.000,C 180.000} C_DIS
LIN {X 104.129,Y 100.316,Z 84.273,A 180.000,B 0.000,C 180.000} C_DIS
LIN {X 104.159,Y 100.244,Z 84.271,A 180.000,B 0.000,C 180.000} C_DIS
LIN {X 104.219,Y 100.100,Z 84.265,A 180.000,B 0.000,C 180.000} C_DIS
LIN {X 104.248,Y 100.027,Z 84.262,A 180.000,B 0.000,C 180.000} C_DIS
LIN {X 104.277,Y 99.955,Z 84.260,A 180.000,B 0.000,C 180.000} C_DIS
LIN {X 104.306,Y 99.883,Z 84.257,A 180.000,B 0.000,C 180.000} C_DIS
LIN {X 104.333,Y 99.810,Z 84.254,A 180.000,B 0.000,C 180.000} C_DIS
LIN {X 104.358,Y 99.737,Z 84.251,A 180.000,B 0.000,C 180.000} C_DIS
LIN {X 104.382,Y 99.664,Z 84.249,A 180.000,B 0.000,C 180.000} C_DIS
LIN {X 104.406,Y 99.591,Z 84.246,A 180.000,B 0.000,C 180.000} C_DIS
LIN {X 104.429,Y 99.518,Z 84.243,A 180.000,B 0.000,C 180.000} C_DIS
LIN {X 104.449,Y 99.444,Z 84.241,A 180.000,B 0.000,C 180.000} C_DIS
LIN {X 104.470,Y 99.368,Z 84.238,A 180.000,B 0.000,C 180.000} C_DIS
LIN {X 104.491,Y 99.293,Z 84.235,A 180.000,B 0.000,C 180.000} C_DIS
LIN {X 104.532,Y 99.141,Z 84.230,A 180.000,B 0.000,C 180.000} C_DIS
LIN {X 104.552,Y 99.067,Z 84.227,A 180.000,B 0.000,C 180.000} C_DIS
LIN {X 104.570,Y 98.992,Z 84.224,A 180.000,B 0.000,C 180.000} C_DIS
LIN {X 104.587,Y 98.917,Z 84.222,A 180.000,B 0.000,C 180.000} C_DIS
LIN {X 104.603,Y 98.842,Z 84.219,A 180.000,B 0.000,C 180.000} C_DIS
LIN {X 104.619,Y 98.765,Z 84.216,A 180.000,B 0.000,C 180.000} C_DIS
LIN {X 104.632,Y 98.689,Z 84.214,A 180.000,B 0.000,C 180.000} C_DIS
LIN {X 104.645,Y 98.612,Z 84.211,A 180.000,B 0.000,C 180.000} C_DIS
LIN {X 104.657,Y 98.535,Z 84.208,A 180.000,B 0.000,C 180.000} C_DIS
LIN {X 104.668,Y 98.458,Z 84.205,A 180.000,B 0.000,C 180.000} C_DIS
LIN {X 104.690,Y 98.303,Z 84.200,A 180.000,B 0.000,C 180.000} C_DIS
LIN {X 104.701,Y 98.226,Z 84.197,A 180.000,B 0.000,C 180.000} C_DIS
LIN {X 104.710,Y 98.149,Z 84.195,A 180.000,B 0.000,C 180.000} C_DIS
LIN {X 104.718,Y 98.072,Z 84.192,A 180.000,B 0.000,C 180.000} C_DIS
LIN {X 104.726,Y 97.995,Z 84.189,A 180.000,B 0.000,C 180.000} C_DIS
LIN {X 104.732,Y 97.918,Z 84.187,A 180.000,B 0.000,C 180.000} C_DIS
LIN {X 104.737,Y 97.841,Z 84.184,A 180.000,B 0.000,C 180.000} C_DIS
LIN {X 104.740,Y 97.763,Z 84.181,A 180.000,B 0.000,C 180.000} C_DIS
LIN {X 104.744,Y 97.685,Z 84.179,A 180.000,B 0.000,C 180.000} C_DIS
LIN {X 104.746,Y 97.607,Z 84.176,A 180.000,B 0.000,C 180.000} C_DIS
LIN {X 104.747,Y 97.529,Z 84.173,A 180.000,B 0.000,C 180.000} C_DIS
LIN {X 104.748,Y 97.450,Z 84.171,A 180.000,B 0.000,C 180.000} C_DIS
LIN {X 104.749,Y 97.372,Z 84.168,A 180.000,B 0.000,C 180.000} C_DIS
LIN {X 104.749,Y 97.293,Z 84.165,A 180.000,B 0.000,C 180.000} C_DIS
LIN {X 104.748,Y 97.216,Z 84.163,A 180.000,B 0.000,C 180.000} C_DIS
LIN {X 104.747,Y 97.138,Z 84.160,A 180.000,B 0.000,C 180.000} C_DIS
LIN {X 104.745,Y 97.061,Z 84.158,A 180.000,B 0.000,C 180.000} C_DIS
LIN {X 104.740,Y 96.983,Z 84.155,A 180.000,B 0.000,C 180.000} C_DIS
LIN {X 104.729,Y 96.828,Z 84.150,A 180.000,B 0.000,C 180.000} C_DIS
LIN {X 104.713,Y 96.673,Z 84.146,A 180.000,B 0.000,C 180.000} C_DIS
LIN {X 104.695,Y 96.517,Z 84.141,A 180.000,B 0.000,C 180.000} C_DIS
LIN {X 104.676,Y 96.362,Z 84.136,A 180.000,B 0.000,C 180.000} C_DIS
LIN {X 104.654,Y 96.207,Z 84.131,A 180.000,B 0.000,C 180.000} C_DIS
LIN {X 104.626,Y 96.053,Z 84.126,A 180.000,B 0.000,C 180.000} C_DIS
LIN {X 104.595,Y 95.901,Z 84.122,A 180.000,B 0.000,C 180.000} C_DIS
LIN {X 104.558,Y 95.749,Z 84.117,A 180.000,B 0.000,C 180.000} C_DIS
LIN {X 104.521,Y 95.597,Z 84.113,A 180.000,B 0.000,C 180.000} C_DIS
LIN {X 104.484,Y 95.445,Z 84.108,A 180.000,B 0.000,C 180.000} C_DIS
LIN {X 104.440,Y 95.294,Z 84.104,A 180.000,B 0.000,C 180.000} C_DIS
LIN {X 104.393,Y 95.144,Z 84.100,A 180.000,B 0.000,C 180.000} C_DIS
LIN {X 104.341,Y 94.997,Z 84.095,A 180.000,B 0.000,C 180.000} C_DIS
LIN {X 104.286,Y 94.851,Z 84.091,A 180.000,B 0.000,C 180.000} C_DIS
LIN {X 104.230,Y 94.705,Z 84.087,A 180.000,B 0.000,C 180.000} C_DIS
LIN {X 104.172,Y 94.559,Z 84.083,A 180.000,B 0.000,C 180.000} C_DIS
LIN {X 104.110,Y 94.416,Z 84.079,A 180.000,B 0.000,C 180.000} C_DIS
LIN {X 104.043,Y 94.274,Z 84.076,A 180.000,B 0.000,C 180.000} C_DIS
LIN {X 103.972,Y 94.134,Z 84.072,A 180.000,B 0.000,C 180.000} C_DIS
LIN {X 103.899,Y 93.995,Z 84.068,A 180.000,B 0.000,C 180.000} C_DIS
LIN {X 103.825,Y 93.857,Z 84.065,A 180.000,B 0.000,C 180.000} C_DIS
LIN {X 103.747,Y 93.720,Z 84.061,A 180.000,B 0.000,C 180.000} C_DIS
LIN {X 103.667,Y 93.585,Z 84.058,A 180.000,B 0.000,C 180.000} C_DIS
LIN {X 103.582,Y 93.454,Z 84.054,A 180.000,B 0.000,C 180.000} C_DIS
LIN {X 103.494,Y 93.324,Z 84.051,A 180.000,B 0.000,C 180.000} C_DIS
LIN {X 103.403,Y 93.196,Z 84.048,A 180.000,B 0.000,C 180.000} C_DIS
LIN {X 103.311,Y 93.069,Z 84.045,A 180.000,B 0.000,C 180.000} C_DIS
LIN {X 103.217,Y 92.943,Z 84.042,A 180.000,B 0.000,C 180.000} C_DIS
LIN {X 103.119,Y 92.820,Z 84.039,A 180.000,B 0.000,C 180.000} C_DIS
LIN {X 103.018,Y 92.700,Z 84.036,A 180.000,B 0.000,C 180.000} C_DIS
LIN {X 102.912,Y 92.583,Z 84.034,A 180.000,B 0.000,C 180.000} C_DIS
LIN {X 102.806,Y 92.468,Z 84.031,A 180.000,B 0.000,C 180.000} C_DIS
LIN {X 102.589,Y 92.240,Z 84.026,A 180.000,B 0.000,C 180.000} C_DIS
LIN {X 102.359,Y 92.026,Z 84.022,A 180.000,B 0.000,C 180.000} C_DIS
LIN {X 102.119,Y 91.822,Z 84.017,A 180.000,B 0.000,C 180.000} C_DIS
LIN {X 101.873,Y 91.625,Z 84.014,A 180.000,B 0.000,C 180.000} C_DIS
LIN {X 101.617,Y 91.443,Z 84.010,A 180.000,B 0.000,C 180.000} C_DIS
LIN {X 101.353,Y 91.271,Z 84.008,A 180.000,B 0.000,C 180.000} C_DIS
LIN {X 101.084,Y 91.107,Z 84.005,A 180.000,B 0.000,C 180.000} C_DIS
LIN {X 100.806,Y 90.960,Z 84.003,A 180.000,B 0.000,C 180.000} C_DIS
LIN {X 100.522,Y 90.824,Z 84.002,A 180.000,B 0.000,C 180.000} C_DIS
LIN {X 100.233,Y 90.698,Z 84.001,A 180.000,B 0.000,C 180.000} C_DIS
LIN {X 99.938,Y 90.588,Z 84.000,A 180.000,B 0.000,C 180.000} C_DIS
LIN {X 99.745,Y 90.525,Z 84.000,A 180.000,B 0.000,C 180.000} C_DIS
; Cutting Move Starts
LIN {X 99.578,Y 90.472,Z 84.000,A 180.000,B 0.000,C 180.000} C_DIS
LIN {X 99.543,Y 90.461,Z 84.000,A 180.000,B 0.000,C 180.000} C_DIS
LIN {X 99.399,Y 90.420,Z 84.000,A 180.000,B 0.000,C 180.000} C_DIS
LIN {X 99.221,Y 90.374,Z 84.000,A 180.000,B 0.000,C 180.000} C_DIS
LIN {X 99.042,Y 90.336,Z 84.000,A 180.000,B 0.000,C 180.000} C_DIS
LIN {X 98.863,Y 90.301,Z 84.000,A 180.000,B 0.000,C 180.000} C_DIS
LIN {X 98.765,Y 90.282,Z 84.000,A 180.000,B 0.000,C 180.000} C_DIS
LIN {X 98.684,Y 90.267,Z 84.000,A 180.000,B 0.000,C 180.000} C_DIS
LIN {X 98.505,Y 90.239,Z 84.000,A 180.000,B 0.000,C 180.000} C_DIS
LIN {X 98.327,Y 90.215,Z 84.000,A 180.000,B 0.000,C 180.000} C_DIS
LIN {X 98.148,Y 90.200,Z 84.000,A 180.000,B 0.000,C 180.000} C_DIS
LIN {X 97.969,Y 90.187,Z 84.000,A 180.000,B 0.000,C 180.000} C_DIS
LIN {X 97.790,Y 90.176,Z 84.000,A 180.000,B 0.000,C 180.000} C_DIS
LIN {X 97.612,Y 90.171,Z 84.000,A 180.000,B 0.000,C 180.000} C_DIS
LIN {X 97.433,Y 90.169,Z 84.000,A 180.000,B 0.000,C 180.000} C_DIS
LIN {X 97.254,Y 90.174,Z 84.000,A 180.000,B 0.000,C 180.000} C_DIS
LIN {X 97.075,Y 90.185,Z 84.000,A 180.000,B 0.000,C 180.000} C_DIS
LIN {X 96.897,Y 90.196,Z 84.000,A 180.000,B 0.000,C 180.000} C_DIS
LIN {X 96.718,Y 90.211,Z 84.000,A 180.000,B 0.000,C 180.000} C_DIS
LIN {X 96.539,Y 90.233,Z 84.000,A 180.000,B 0.000,C 180.000} C_DIS
LIN {X 96.360,Y 90.259,Z 84.000,A 180.000,B 0.000,C 180.000} C_DIS
LIN {X 96.235,Y 90.282,Z 84.000,A 180.000,B 0.000,C 180.000} C_DIS
LIN {X 96.181,Y 90.292,Z 84.000,A 180.000,B 0.000,C 180.000} C_DIS
LIN {X 96.003,Y 90.327,Z 84.000,A 180.000,B 0.000,C 180.000} C_DIS
LIN {X 95.824,Y 90.363,Z 84.000,A 180.000,B 0.000,C 180.000} C_DIS
LIN {X 95.645,Y 90.408,Z 84.000,A 180.000,B 0.000,C 180.000} C_DIS
LIN {X 95.466,Y 90.458,Z 84.000,A 180.000,B 0.000,C 180.000} C_DIS
LIN {X 95.457,Y 90.461,Z 84.000,A 180.000,B 0.000,C 180.000} C_DIS
LIN {X 95.288,Y 90.515,Z 84.000,A 180.000,B 0.000,C 180.000} C_DIS
LIN {X 95.109,Y 90.573,Z 84.000,A 180.000,B 0.000,C 180.000} C_DIS
LIN {X 94.930,Y 90.635,Z 84.000,A 180.000,B 0.000,C 180.000} C_DIS
LIN {X 94.918,Y 90.640,Z 84.000,A 180.000,B 0.000,C 180.000} C_DIS
LIN {X 94.751,Y 90.703,Z 84.000,A 180.000,B 0.000,C 180.000} C_DIS
LIN {X 94.573,Y 90.781,Z 84.000,A 180.000,B 0.000,C 180.000} C_DIS
LIN {X 94.490,Y 90.818,Z 84.000,A 180.000,B 0.000,C 180.000} C_DIS
LIN {X 94.394,Y 90.863,Z 84.000,A 180.000,B 0.000,C 180.000} C_DIS
LIN {X 94.215,Y 90.948,Z 84.000,A 180.000,B 0.000,C 180.000} C_DIS
LIN {X 94.118,Y 90.997,Z 84.000,A 180.000,B 0.000,C 180.000} C_DIS
LIN {X 94.036,Y 91.039,Z 84.000,A 180.000,B 0.000,C 180.000} C_DIS
LIN {X 93.857,Y 91.139,Z 84.000,A 180.000,B 0.000,C 180.000} C_DIS
LIN {X 93.795,Y 91.176,Z 84.000,A 180.000,B 0.000,C 180.000} C_DIS
LIN {X 93.679,Y 91.246,Z 84.000,A 180.000,B 0.000,C 180.000} C_DIS
LIN {X 93.500,Y 91.360,Z 84.000,A 180.000,B 0.000,C 180.000} C_DIS
LIN {X 93.321,Y 91.478,Z 84.000,A 180.000,B 0.000,C 180.000} C_DIS
LIN {X 93.240,Y 91.533,Z 84.000,A 180.000,B 0.000,C 180.000} C_DIS
LIN {X 93.142,Y 91.605,Z 84.000,A 180.000,B 0.000,C 180.000} C_DIS
LIN {X 93.002,Y 91.712,Z 84.000,A 180.000,B 0.000,C 180.000} C_DIS
LIN {X 92.964,Y 91.743,Z 84.000,A 180.000,B 0.000,C 180.000} C_DIS
LIN {X 92.785,Y 91.891,Z 84.000,A 180.000,B 0.000,C 180.000} C_DIS
LIN {X 92.606,Y 92.042,Z 84.000,A 180.000,B 0.000,C 180.000} C_DIS
LIN {X 92.575,Y 92.070,Z 84.000,A 180.000,B 0.000,C 180.000} C_DIS
LIN {X 92.427,Y 92.208,Z 84.000,A 180.000,B 0.000,C 180.000} C_DIS
LIN {X 92.385,Y 92.249,Z 84.000,A 180.000,B 0.000,C 180.000} C_DIS
LIN {X 92.249,Y 92.389,Z 84.000,A 180.000,B 0.000,C 180.000} C_DIS
LIN {X 92.213,Y 92.427,Z 84.000,A 180.000,B 0.000,C 180.000} C_DIS
LIN {X 92.070,Y 92.579,Z 84.000,A 180.000,B 0.000,C 180.000} C_DIS
LIN {X 92.045,Y 92.606,Z 84.000,A 180.000,B 0.000,C 180.000} C_DIS
LIN {X 91.891,Y 92.781,Z 84.000,A 180.000,B 0.000,C 180.000} C_DIS
LIN {X 91.887,Y 92.785,Z 84.000,A 180.000,B 0.000,C 180.000} C_DIS
LIN {X 91.742,Y 92.964,Z 84.000,A 180.000,B 0.000,C 180.000} C_DIS
LIN {X 91.712,Y 93.003,Z 84.000,A 180.000,B 0.000,C 180.000} C_DIS
LIN {X 91.609,Y 93.142,Z 84.000,A 180.000,B 0.000,C 180.000} C_DIS
LIN {X 91.479,Y 93.321,Z 84.000,A 180.000,B 0.000,C 180.000} C_DIS
LIN {X 91.357,Y 93.500,Z 84.000,A 180.000,B 0.000,C 180.000} C_DIS
LIN {X 91.355,Y 93.504,Z 84.000,A 180.000,B 0.000,C 180.000} C_DIS
LIN {X 91.245,Y 93.679,Z 84.000,A 180.000,B 0.000,C 180.000} C_DIS
LIN {X 91.176,Y 93.795,Z 84.000,A 180.000,B 0.000,C 180.000} C_DIS
LIN {X 91.140,Y 93.857,Z 84.000,A 180.000,B 0.000,C 180.000} C_DIS
LIN {X 91.042,Y 94.036,Z 84.000,A 180.000,B 0.000,C 180.000} C_DIS
LIN {X 90.997,Y 94.119,Z 84.000,A 180.000,B 0.000,C 180.000} C_DIS
LIN {X 90.948,Y 94.215,Z 84.000,A 180.000,B 0.000,C 180.000} C_DIS
LIN {X 90.860,Y 94.394,Z 84.000,A 180.000,B 0.000,C 180.000} C_DIS
LIN {X 90.818,Y 94.486,Z 84.000,A 180.000,B 0.000,C 180.000} C_DIS
LIN {X 90.780,Y 94.573,Z 84.000,A 180.000,B 0.000,C 180.000} C_DIS
LIN {X 90.707,Y 94.751,Z 84.000,A 180.000,B 0.000,C 180.000} C_DIS
LIN {X 90.640,Y 94.924,Z 84.000,A 180.000,B 0.000,C 180.000} C_DIS
LIN {X 90.637,Y 94.930,Z 84.000,A 180.000,B 0.000,C 180.000} C_DIS
LIN {X 90.570,Y 95.109,Z 84.000,A 180.000,B 0.000,C 180.000} C_DIS
LIN {X 90.511,Y 95.288,Z 84.000,A 180.000,B 0.000,C 180.000} C_DIS
LIN {X 90.461,Y 95.456,Z 84.000,A 180.000,B 0.000,C 180.000} C_DIS
LIN {X 90.458,Y 95.466,Z 84.000,A 180.000,B 0.000,C 180.000} C_DIS
LIN {X 90.412,Y 95.645,Z 84.000,A 180.000,B 0.000,C 180.000} C_DIS
LIN {X 90.366,Y 95.824,Z 84.000,A 180.000,B 0.000,C 180.000} C_DIS
LIN {X 90.324,Y 96.003,Z 84.000,A 180.000,B 0.000,C 180.000} C_DIS
LIN {X 90.288,Y 96.181,Z 84.000,A 180.000,B 0.000,C 180.000} C_DIS
LIN {X 90.282,Y 96.216,Z 84.000,A 180.000,B 0.000,C 180.000} C_DIS
LIN {X 90.260,Y 96.360,Z 84.000,A 180.000,B 0.000,C 180.000} C_DIS
LIN {X 90.236,Y 96.539,Z 84.000,A 180.000,B 0.000,C 180.000} C_DIS
LIN {X 90.218,Y 96.681,Z 84.000,A 180.000,B 0.000,C 180.000} C_DIS
LIN {X 90.213,Y 96.718,Z 84.000,A 180.000,B 0.000,C 180.000} C_DIS
LIN {X 90.195,Y 96.897,Z 84.000,A 180.000,B 0.000,C 180.000} C_DIS
LIN {X 90.181,Y 97.075,Z 84.000,A 180.000,B 0.000,C 180.000} C_DIS
LIN {X 90.175,Y 97.254,Z 84.000,A 180.000,B 0.000,C 180.000} C_DIS
LIN {X 90.172,Y 97.433,Z 84.000,A 180.000,B 0.000,C 180.000} C_DIS
LIN {X 90.172,Y 97.612,Z 84.000,A 180.000,B 0.000,C 180.000} C_DIS
LIN {X 90.176,Y 97.790,Z 84.000,A 180.000,B 0.000,C 180.000} C_DIS
LIN {X 90.184,Y 97.969,Z 84.000,A 180.000,B 0.000,C 180.000} C_DIS
LIN {X 90.199,Y 98.148,Z 84.000,A 180.000,B 0.000,C 180.000} C_DIS
LIN {X 90.219,Y 98.327,Z 84.000,A 180.000,B 0.000,C 180.000} C_DIS
LIN {X 90.241,Y 98.505,Z 84.000,A 180.000,B 0.000,C 180.000} C_DIS
LIN {X 90.266,Y 98.684,Z 84.000,A 180.000,B 0.000,C 180.000} C_DIS
LIN {X 90.282,Y 98.784,Z 84.000,A 180.000,B 0.000,C 180.000} C_DIS
LIN {X 90.297,Y 98.863,Z 84.000,A 180.000,B 0.000,C 180.000} C_DIS
LIN {X 90.333,Y 99.042,Z 84.000,A 180.000,B 0.000,C 180.000} C_DIS
LIN {X 90.377,Y 99.221,Z 84.000,A 180.000,B 0.000,C 180.000} C_DIS
LIN {X 90.423,Y 99.399,Z 84.000,A 180.000,B 0.000,C 180.000} C_DIS
LIN {X 90.461,Y 99.544,Z 84.000,A 180.000,B 0.000,C 180.000} C_DIS
LIN {X 90.470,Y 99.578,Z 84.000,A 180.000,B 0.000,C 180.000} C_DIS
LIN {X 90.526,Y 99.757,Z 84.000,A 180.000,B 0.000,C 180.000} C_DIS
LIN {X 90.586,Y 99.936,Z 84.000,A 180.000,B 0.000,C 180.000} C_DIS
LIN {X 90.640,Y 100.076,Z 84.000,A 180.000,B 0.000,C 180.000} C_DIS
LIN {X 90.654,Y 100.114,Z 84.000,A 180.000,B 0.000,C 180.000} C_DIS
LIN {X 90.725,Y 100.293,Z 84.000,A 180.000,B 0.000,C 180.000} C_DIS
LIN {X 90.799,Y 100.472,Z 84.000,A 180.000,B 0.000,C 180.000} C_DIS
LIN {X 90.818,Y 100.514,Z 84.000,A 180.000,B 0.000,C 180.000} C_DIS
LIN {X 90.880,Y 100.651,Z 84.000,A 180.000,B 0.000,C 180.000} C_DIS
LIN {X 90.971,Y 100.829,Z 84.000,A 180.000,B 0.000,C 180.000} C_DIS
LIN {X 90.997,Y 100.881,Z 84.000,A 180.000,B 0.000,C 180.000} C_DIS
LIN {X 91.067,Y 101.008,Z 84.000,A 180.000,B 0.000,C 180.000} C_DIS
LIN {X 91.166,Y 101.187,Z 84.000,A 180.000,B 0.000,C 180.000} C_DIS
LIN {X 91.176,Y 101.205,Z 84.000,A 180.000,B 0.000,C 180.000} C_DIS
LIN {X 91.271,Y 101.366,Z 84.000,A 180.000,B 0.000,C 180.000} C_DIS
LIN {X 91.355,Y 101.496,Z 84.000,A 180.000,B 0.000,C 180.000} C_DIS
LIN {X 91.387,Y 101.545,Z 84.000,A 180.000,B 0.000,C 180.000} C_DIS
LIN {X 91.511,Y 101.723,Z 84.000,A 180.000,B 0.000,C 180.000} C_DIS
LIN {X 91.533,Y 101.754,Z 84.000,A 180.000,B 0.000,C 180.000} C_DIS
LIN {X 91.641,Y 101.902,Z 84.000,A 180.000,B 0.000,C 180.000} C_DIS
LIN {X 91.712,Y 101.997,Z 84.000,A 180.000,B 0.000,C 180.000} C_DIS
LIN {X 91.776,Y 102.081,Z 84.000,A 180.000,B 0.000,C 180.000} C_DIS
LIN {X 91.891,Y 102.219,Z 84.000,A 180.000,B 0.000,C 180.000} C_DIS
LIN {X 91.925,Y 102.260,Z 84.000,A 180.000,B 0.000,C 180.000} C_DIS
LIN {X 92.070,Y 102.421,Z 84.000,A 180.000,B 0.000,C 180.000} C_DIS
LIN {X 92.086,Y 102.438,Z 84.000,A 180.000,B 0.000,C 180.000} C_DIS
LIN {X 92.249,Y 102.611,Z 84.000,A 180.000,B 0.000,C 180.000} C_DIS
LIN {X 92.255,Y 102.617,Z 84.000,A 180.000,B 0.000,C 180.000} C_DIS
LIN {X 92.427,Y 102.792,Z 84.000,A 180.000,B 0.000,C 180.000} C_DIS
LIN {X 92.432,Y 102.796,Z 84.000,A 180.000,B 0.000,C 180.000} C_DIS
LIN {X 92.606,Y 102.958,Z 84.000,A 180.000,B 0.000,C 180.000} C_DIS
LIN {X 92.626,Y 102.975,Z 84.000,A 180.000,B 0.000,C 180.000} C_DIS
LIN {X 92.785,Y 103.109,Z 84.000,A 180.000,B 0.000,C 180.000} C_DIS
LIN {X 92.964,Y 103.257,Z 84.000,A 180.000,B 0.000,C 180.000} C_DIS
LIN {X 93.060,Y 103.332,Z 84.000,A 180.000,B 0.000,C 180.000} C_DIS
LIN {X 93.142,Y 103.395,Z 84.000,A 180.000,B 0.000,C 180.000} C_DIS
LIN {X 93.304,Y 103.511,Z 84.000,A 180.000,B 0.000,C 180.000} C_DIS
LIN {X 93.321,Y 103.522,Z 84.000,A 180.000,B 0.000,C 180.000} C_DIS
LIN {X 93.500,Y 103.640,Z 84.000,A 180.000,B 0.000,C 180.000} C_DIS
LIN {X 93.679,Y 103.754,Z 84.000,A 180.000,B 0.000,C 180.000} C_DIS
LIN {X 93.857,Y 103.861,Z 84.000,A 180.000,B 0.000,C 180.000} C_DIS
LIN {X 93.870,Y 103.869,Z 84.000,A 180.000,B 0.000,C 180.000} C_DIS
LIN {X 94.036,Y 103.961,Z 84.000,A 180.000,B 0.000,C 180.000} C_DIS
LIN {X 94.205,Y 104.047,Z 84.000,A 180.000,B 0.000,C 180.000} C_DIS
LIN {X 94.215,Y 104.052,Z 84.000,A 180.000,B 0.000,C 180.000} C_DIS
LIN {X 94.394,Y 104.137,Z 84.000,A 180.000,B 0.000,C 180.000} C_DIS
LIN {X 94.573,Y 104.219,Z 84.000,A 180.000,B 0.000,C 180.000} C_DIS
LIN {X 94.589,Y 104.226,Z 84.000,A 180.000,B 0.000,C 180.000} C_DIS
LIN {X 94.751,Y 104.297,Z 84.000,A 180.000,B 0.000,C 180.000} C_DIS
LIN {X 94.930,Y 104.365,Z 84.000,A 180.000,B 0.000,C 180.000} C_DIS
LIN {X 95.041,Y 104.405,Z 84.000,A 180.000,B 0.000,C 180.000} C_DIS
LIN {X 95.109,Y 104.427,Z 84.000,A 180.000,B 0.000,C 180.000} C_DIS
LIN {X 95.288,Y 104.485,Z 84.000,A 180.000,B 0.000,C 180.000} C_DIS
LIN {X 95.466,Y 104.542,Z 84.000,A 180.000,B 0.000,C 180.000} C_DIS
LIN {X 95.613,Y 104.584,Z 84.000,A 180.000,B 0.000,C 180.000} C_DIS
LIN {X 95.645,Y 104.592,Z 84.000,A 180.000,B 0.000,C 180.000} C_DIS
LIN {X 95.824,Y 104.637,Z 84.000,A 180.000,B 0.000,C 180.000} C_DIS
LIN {X 96.003,Y 104.673,Z 84.000,A 180.000,B 0.000,C 180.000} C_DIS
LIN {X 96.181,Y 104.708,Z 84.000,A 180.000,B 0.000,C 180.000} C_DIS
LIN {X 96.360,Y 104.741,Z 84.000,A 180.000,B 0.000,C 180.000} C_DIS
LIN {X 96.505,Y 104.762,Z 84.000,A 180.000,B 0.000,C 180.000} C_DIS
LIN {X 96.539,Y 104.767,Z 84.000,A 180.000,B 0.000,C 180.000} C_DIS
LIN {X 96.718,Y 104.789,Z 84.000,A 180.000,B 0.000,C 180.000} C_DIS
LIN {X 96.897,Y 104.804,Z 84.000,A 180.000,B 0.000,C 180.000} C_DIS
LIN {X 97.075,Y 104.815,Z 84.000,A 180.000,B 0.000,C 180.000} C_DIS
LIN {X 97.254,Y 104.826,Z 84.000,A 180.000,B 0.000,C 180.000} C_DIS
LIN {X 97.433,Y 104.831,Z 84.000,A 180.000,B 0.000,C 180.000} C_DIS
LIN {X 97.612,Y 104.829,Z 84.000,A 180.000,B 0.000,C 180.000} C_DIS
LIN {X 97.790,Y 104.824,Z 84.000,A 180.000,B 0.000,C 180.000} C_DIS
LIN {X 97.969,Y 104.813,Z 84.000,A 180.000,B 0.000,C 180.000} C_DIS
LIN {X 98.148,Y 104.800,Z 84.000,A 180.000,B 0.000,C 180.000} C_DIS
LIN {X 98.327,Y 104.785,Z 84.000,A 180.000,B 0.000,C 180.000} C_DIS
LIN {X 98.495,Y 104.762,Z 84.000,A 180.000,B 0.000,C 180.000} C_DIS
LIN {X 98.505,Y 104.761,Z 84.000,A 180.000,B 0.000,C 180.000} C_DIS
LIN {X 98.684,Y 104.733,Z 84.000,A 180.000,B 0.000,C 180.000} C_DIS
LIN {X 98.863,Y 104.699,Z 84.000,A 180.000,B 0.000,C 180.000} C_DIS
LIN {X 99.042,Y 104.664,Z 84.000,A 180.000,B 0.000,C 180.000} C_DIS
LIN {X 99.221,Y 104.626,Z 84.000,A 180.000,B 0.000,C 180.000} C_DIS
LIN {X 99.387,Y 104.584,Z 84.000,A 180.000,B 0.000,C 180.000} C_DIS
LIN {X 99.399,Y 104.580,Z 84.000,A 180.000,B 0.000,C 180.000} C_DIS
LIN {X 99.578,Y 104.528,Z 84.000,A 180.000,B 0.000,C 180.000} C_DIS
LIN {X 99.757,Y 104.471,Z 84.000,A 180.000,B 0.000,C 180.000} C_DIS
LIN {X 99.936,Y 104.413,Z 84.000,A 180.000,B 0.000,C 180.000} C_DIS
LIN {X 99.959,Y 104.405,Z 84.000,A 180.000,B 0.000,C 180.000} C_DIS
LIN {X 100.114,Y 104.348,Z 84.000,A 180.000,B 0.000,C 180.000} C_DIS
LIN {X 100.293,Y 104.278,Z 84.000,A 180.000,B 0.000,C 180.000} C_DIS
LIN {X 100.411,Y 104.226,Z 84.000,A 180.000,B 0.000,C 180.000} C_DIS
LIN {X 100.472,Y 104.199,Z 84.000,A 180.000,B 0.000,C 180.000} C_DIS
LIN {X 100.651,Y 104.116,Z 84.000,A 180.000,B 0.000,C 180.000} C_DIS
LIN {X 100.795,Y 104.047,Z 84.000,A 180.000,B 0.000,C 180.000} C_DIS
LIN {X 100.829,Y 104.030,Z 84.000,A 180.000,B 0.000,C 180.000} C_DIS
LIN {X 101.008,Y 103.937,Z 84.000,A 180.000,B 0.000,C 180.000} C_DIS
LIN {X 101.130,Y 103.869,Z 84.000,A 180.000,B 0.000,C 180.000} C_DIS
LIN {X 101.187,Y 103.835,Z 84.000,A 180.000,B 0.000,C 180.000} C_DIS
LIN {X 101.366,Y 103.725,Z 84.000,A 180.000,B 0.000,C 180.000} C_DIS
LIN {X 101.422,Y 103.690,Z 84.000,A 180.000,B 0.000,C 180.000} C_DIS
LIN {X 101.545,Y 103.612,Z 84.000,A 180.000,B 0.000,C 180.000} C_DIS
LIN {X 101.696,Y 103.511,Z 84.000,A 180.000,B 0.000,C 180.000} C_DIS
LIN {X 101.723,Y 103.492,Z 84.000,A 180.000,B 0.000,C 180.000} C_DIS
LIN {X 101.902,Y 103.361,Z 84.000,A 180.000,B 0.000,C 180.000} C_DIS
LIN {X 101.940,Y 103.332,Z 84.000,A 180.000,B 0.000,C 180.000} C_DIS
LIN {X 102.081,Y 103.220,Z 84.000,A 180.000,B 0.000,C 180.000} C_DIS
LIN {X 102.161,Y 103.153,Z 84.000,A 180.000,B 0.000,C 180.000} C_DIS
LIN {X 102.260,Y 103.072,Z 84.000,A 180.000,B 0.000,C 180.000} C_DIS
LIN {X 102.374,Y 102.975,Z 84.000,A 180.000,B 0.000,C 180.000} C_DIS
LIN {X 102.438,Y 102.918,Z 84.000,A 180.000,B 0.000,C 180.000} C_DIS
LIN {X 102.568,Y 102.796,Z 84.000,A 180.000,B 0.000,C 180.000} C_DIS
LIN {X 102.617,Y 102.750,Z 84.000,A 180.000,B 0.000,C 180.000} C_DIS
LIN {X 102.745,Y 102.617,Z 84.000,A 180.000,B 0.000,C 180.000} C_DIS
LIN {X 102.796,Y 102.564,Z 84.000,A 180.000,B 0.000,C 180.000} C_DIS
LIN {X 102.914,Y 102.438,Z 84.000,A 180.000,B 0.000,C 180.000} C_DIS
LIN {X 102.975,Y 102.373,Z 84.000,A 180.000,B 0.000,C 180.000} C_DIS
LIN {X 103.075,Y 102.260,Z 84.000,A 180.000,B 0.000,C 180.000} C_DIS
LIN {X 103.153,Y 102.167,Z 84.000,A 180.000,B 0.000,C 180.000} C_DIS
LIN {X 103.224,Y 102.081,Z 84.000,A 180.000,B 0.000,C 180.000} C_DIS
LIN {X 103.332,Y 101.937,Z 84.000,A 180.000,B 0.000,C 180.000} C_DIS
LIN {X 103.359,Y 101.902,Z 84.000,A 180.000,B 0.000,C 180.000} C_DIS
LIN {X 103.489,Y 101.723,Z 84.000,A 180.000,B 0.000,C 180.000} C_DIS
LIN {X 103.511,Y 101.693,Z 84.000,A 180.000,B 0.000,C 180.000} C_DIS
LIN {X 103.613,Y 101.545,Z 84.000,A 180.000,B 0.000,C 180.000} C_DIS
LIN {X 103.690,Y 101.429,Z 84.000,A 180.000,B 0.000,C 180.000} C_DIS
LIN {X 103.729,Y 101.366,Z 84.000,A 180.000,B 0.000,C 180.000} C_DIS
LIN {X 103.834,Y 101.187,Z 84.000,A 180.000,B 0.000,C 180.000} C_DIS
LIN {X 103.869,Y 101.126,Z 84.000,A 180.000,B 0.000,C 180.000} C_DIS
LIN {X 103.933,Y 101.008,Z 84.000,A 180.000,B 0.000,C 180.000} C_DIS
LIN {X 104.029,Y 100.829,Z 84.000,A 180.000,B 0.000,C 180.000} C_DIS
LIN {X 104.047,Y 100.795,Z 84.000,A 180.000,B 0.000,C 180.000} C_DIS
LIN {X 104.120,Y 100.651,Z 84.000,A 180.000,B 0.000,C 180.000} C_DIS
LIN {X 104.201,Y 100.472,Z 84.000,A 180.000,B 0.000,C 180.000} C_DIS
LIN {X 104.226,Y 100.414,Z 84.000,A 180.000,B 0.000,C 180.000} C_DIS
LIN {X 104.275,Y 100.293,Z 84.000,A 180.000,B 0.000,C 180.000} C_DIS
LIN {X 104.346,Y 100.114,Z 84.000,A 180.000,B 0.000,C 180.000} C_DIS
LIN {X 104.405,Y 99.959,Z 84.000,A 180.000,B 0.000,C 180.000} C_DIS
LIN {X 104.414,Y 99.936,Z 84.000,A 180.000,B 0.000,C 180.000} C_DIS
LIN {X 104.474,Y 99.757,Z 84.000,A 180.000,B 0.000,C 180.000} C_DIS
LIN {X 104.530,Y 99.578,Z 84.000,A 180.000,B 0.000,C 180.000} C_DIS
LIN {X 104.577,Y 99.399,Z 84.000,A 180.000,B 0.000,C 180.000} C_DIS
LIN {X 104.584,Y 99.372,Z 84.000,A 180.000,B 0.000,C 180.000} C_DIS
LIN {X 104.623,Y 99.221,Z 84.000,A 180.000,B 0.000,C 180.000} C_DIS
LIN {X 104.667,Y 99.042,Z 84.000,A 180.000,B 0.000,C 180.000} C_DIS
LIN {X 104.703,Y 98.863,Z 84.000,A 180.000,B 0.000,C 180.000} C_DIS
LIN {X 104.734,Y 98.684,Z 84.000,A 180.000,B 0.000,C 180.000} C_DIS
LIN {X 104.759,Y 98.505,Z 84.000,A 180.000,B 0.000,C 180.000} C_DIS
LIN {X 104.762,Y 98.476,Z 84.000,A 180.000,B 0.000,C 180.000} C_DIS
LIN {X 104.781,Y 98.327,Z 84.000,A 180.000,B 0.000,C 180.000} C_DIS
LIN {X 104.801,Y 98.148,Z 84.000,A 180.000,B 0.000,C 180.000} C_DIS
LIN {X 104.816,Y 97.969,Z 84.000,A 180.000,B 0.000,C 180.000} C_DIS
LIN {X 104.824,Y 97.790,Z 84.000,A 180.000,B 0.000,C 180.000} C_DIS
LIN {X 104.828,Y 97.612,Z 84.000,A 180.000,B 0.000,C 180.000} C_DIS
LIN {X 104.828,Y 97.433,Z 84.000,A 180.000,B 0.000,C 180.000} C_DIS
LIN {X 104.825,Y 97.254,Z 84.000,A 180.000,B 0.000,C 180.000} C_DIS
LIN {X 104.819,Y 97.075,Z 84.000,A 180.000,B 0.000,C 180.000} C_DIS
LIN {X 104.805,Y 96.897,Z 84.000,A 180.000,B 0.000,C 180.000} C_DIS
LIN {X 104.787,Y 96.718,Z 84.000,A 180.000,B 0.000,C 180.000} C_DIS
LIN {X 104.762,Y 96.524,Z 84.000,A 180.000,B 0.000,C 180.000} C_DIS
LIN {X 104.740,Y 96.360,Z 84.000,A 180.000,B 0.000,C 180.000} C_DIS
LIN {X 104.712,Y 96.181,Z 84.000,A 180.000,B 0.000,C 180.000} C_DIS
LIN {X 104.676,Y 96.003,Z 84.000,A 180.000,B 0.000,C 180.000} C_DIS
LIN {X 104.634,Y 95.824,Z 84.000,A 180.000,B 0.000,C 180.000} C_DIS
LIN {X 104.588,Y 95.645,Z 84.000,A 180.000,B 0.000,C 180.000} C_DIS
LIN {X 104.584,Y 95.628,Z 84.000,A 180.000,B 0.000,C 180.000} C_DIS
LIN {X 104.542,Y 95.466,Z 84.000,A 180.000,B 0.000,C 180.000} C_DIS
LIN {X 104.489,Y 95.288,Z 84.000,A 180.000,B 0.000,C 180.000} C_DIS
LIN {X 104.430,Y 95.109,Z 84.000,A 180.000,B 0.000,C 180.000} C_DIS
LIN {X 104.405,Y 95.041,Z 84.000,A 180.000,B 0.000,C 180.000} C_DIS
LIN {X 104.363,Y 94.930,Z 84.000,A 180.000,B 0.000,C 180.000} C_DIS
LIN {X 104.293,Y 94.751,Z 84.000,A 180.000,B 0.000,C 180.000} C_DIS
LIN {X 104.226,Y 94.586,Z 84.000,A 180.000,B 0.000,C 180.000} C_DIS
LIN {X 104.220,Y 94.573,Z 84.000,A 180.000,B 0.000,C 180.000} C_DIS
LIN {X 104.140,Y 94.394,Z 84.000,A 180.000,B 0.000,C 180.000} C_DIS
LIN {X 104.052,Y 94.215,Z 84.000,A 180.000,B 0.000,C 180.000} C_DIS
LIN {X 104.047,Y 94.205,Z 84.000,A 180.000,B 0.000,C 180.000} C_DIS
LIN {X 103.958,Y 94.036,Z 84.000,A 180.000,B 0.000,C 180.000} C_DIS
LIN {X 103.860,Y 93.857,Z 84.000,A 180.000,B 0.000,C 180.000} C_DIS
LIN {X 103.755,Y 93.679,Z 84.000,A 180.000,B 0.000,C 180.000} C_DIS
LIN {X 103.690,Y 93.571,Z 84.000,A 180.000,B 0.000,C 180.000} C_DIS
LIN {X 103.643,Y 93.500,Z 84.000,A 180.000,B 0.000,C 180.000} C_DIS
LIN {X 103.521,Y 93.321,Z 84.000,A 180.000,B 0.000,C 180.000} C_DIS
LIN {X 103.511,Y 93.307,Z 84.000,A 180.000,B 0.000,C 180.000} C_DIS
LIN {X 103.391,Y 93.142,Z 84.000,A 180.000,B 0.000,C 180.000} C_DIS
LIN {X 103.332,Y 93.063,Z 84.000,A 180.000,B 0.000,C 180.000} C_DIS
LIN {X 103.258,Y 92.964,Z 84.000,A 180.000,B 0.000,C 180.000} C_DIS
LIN {X 103.153,Y 92.833,Z 84.000,A 180.000,B 0.000,C 180.000} C_DIS
LIN {X 103.113,Y 92.785,Z 84.000,A 180.000,B 0.000,C 180.000} C_DIS
LIN {X 102.975,Y 92.627,Z 84.000,A 180.000,B 0.000,C 180.000} C_DIS
LIN {X 102.955,Y 92.606,Z 84.000,A 180.000,B 0.000,C 180.000} C_DIS
LIN {X 102.796,Y 92.436,Z 84.000,A 180.000,B 0.000,C 180.000} C_DIS
LIN {X 102.787,Y 92.427,Z 84.000,A 180.000,B 0.000,C 180.000} C_DIS
LIN {X 102.617,Y 92.250,Z 84.000,A 180.000,B 0.000,C 180.000} C_DIS
LIN {X 102.615,Y 92.249,Z 84.000,A 180.000,B 0.000,C 180.000} C_DIS
LIN {X 102.438,Y 92.082,Z 84.000,A 180.000,B 0.000,C 180.000} C_DIS
LIN {X 102.425,Y 92.070,Z 84.000,A 180.000,B 0.000,C 180.000} C_DIS
LIN {X 102.260,Y 91.928,Z 84.000,A 180.000,B 0.000,C 180.000} C_DIS
LIN {X 102.215,Y 91.891,Z 84.000,A 180.000,B 0.000,C 180.000} C_DIS
LIN {X 102.081,Y 91.780,Z 84.000,A 180.000,B 0.000,C 180.000} C_DIS
LIN {X 101.998,Y 91.712,Z 84.000,A 180.000,B 0.000,C 180.000} C_DIS
LIN {X 101.902,Y 91.639,Z 84.000,A 180.000,B 0.000,C 180.000} C_DIS
LIN {X 101.760,Y 91.533,Z 84.000,A 180.000,B 0.000,C 180.000} C_DIS
LIN {X 101.723,Y 91.508,Z 84.000,A 180.000,B 0.000,C 180.000} C_DIS
LIN {X 101.545,Y 91.388,Z 84.000,A 180.000,B 0.000,C 180.000} C_DIS
LIN {X 101.492,Y 91.355,Z 84.000,A 180.000,B 0.000,C 180.000} C_DIS
LIN {X 101.366,Y 91.275,Z 84.000,A 180.000,B 0.000,C 180.000} C_DIS
LIN {X 101.205,Y 91.176,Z 84.000,A 180.000,B 0.000,C 180.000} C_DIS
LIN {X 101.187,Y 91.165,Z 84.000,A 180.000,B 0.000,C 180.000} C_DIS
LIN {X 101.008,Y 91.063,Z 84.000,A 180.000,B 0.000,C 180.000} C_DIS
LIN {X 100.882,Y 90.997,Z 84.000,A 180.000,B 0.000,C 180.000} C_DIS
LIN {X 100.829,Y 90.970,Z 84.000,A 180.000,B 0.000,C 180.000} C_DIS
LIN {X 100.651,Y 90.884,Z 84.000,A 180.000,B 0.000,C 180.000} C_DIS
LIN {X 100.510,Y 90.818,Z 84.000,A 180.000,B 0.000,C 180.000} C_DIS
LIN {X 100.472,Y 90.801,Z 84.000,A 180.000,B 0.000,C 180.000} C_DIS
LIN {X 100.293,Y 90.722,Z 84.000,A 180.000,B 0.000,C 180.000} C_DIS
LIN {X 100.114,Y 90.652,Z 84.000,A 180.000,B 0.000,C 180.000} C_DIS
LIN {X 100.082,Y 90.640,Z 84.000,A 180.000,B 0.000,C 180.000} C_DIS
LIN {X 99.936,Y 90.587,Z 84.000,A 180.000,B 0.000,C 180.000} C_DIS
LIN {X 99.757,Y 90.529,Z 84.000,A 180.000,B 0.000,C 180.000} C_DIS
LIN {X 99.745,Y 90.525,Z 84.000,A 180.000,B 0.000,C 180.000} C_DIS
; Link Move Starts
LIN {X 99.451,Y 90.433,Z 84.000,A 180.000,B 0.000,C 180.000} C_DIS
LIN {X 99.178,Y 90.363,Z 83.999,A 180.000,B 0.000,C 180.000} C_DIS
LIN {X 98.885,Y 90.304,Z 83.998,A 180.000,B 0.000,C 180.000} C_DIS
LIN {X 98.598,Y 90.251,Z 83.997,A 180.000,B 0.000,C 180.000} C_DIS
LIN {X 98.296,Y 90.210,Z 83.995,A 180.000,B 0.000,C 180.000} C_DIS
LIN {X 98.005,Y 90.186,Z 83.992,A 180.000,B 0.000,C 180.000} C_DIS
LIN {X 97.709,Y 90.169,Z 83.990,A 180.000,B 0.000,C 180.000} C_DIS
LIN {X 97.420,Y 90.163,Z 83.987,A 180.000,B 0.000,C 180.000} C_DIS
LIN {X 97.115,Y 90.174,Z 83.983,A 180.000,B 0.000,C 180.000} C_DIS
LIN {X 96.816,Y 90.193,Z 83.979,A 180.000,B 0.000,C 180.000} C_DIS
LIN {X 96.528,Y 90.223,Z 83.975,A 180.000,B 0.000,C 180.000} C_DIS
LIN {X 96.239,Y 90.267,Z 83.971,A 180.000,B 0.000,C 180.000} C_DIS
LIN {X 96.085,Y 90.295,Z 83.968,A 180.000,B 0.000,C 180.000} C_DIS
LIN {X 95.932,Y 90.324,Z 83.965,A 180.000,B 0.000,C 180.000} C_DIS
LIN {X 95.790,Y 90.353,Z 83.963,A 180.000,B 0.000,C 180.000} C_DIS
LIN {X 95.650,Y 90.388,Z 83.960,A 180.000,B 0.000,C 180.000} C_DIS
LIN {X 95.509,Y 90.424,Z 83.957,A 180.000,B 0.000,C 180.000} C_DIS
LIN {X 95.371,Y 90.466,Z 83.955,A 180.000,B 0.000,C 180.000} C_DIS
LIN {X 95.222,Y 90.512,Z 83.952,A 180.000,B 0.000,C 180.000} C_DIS
LIN {X 95.073,Y 90.559,Z 83.948,A 180.000,B 0.000,C 180.000} C_DIS
LIN {X 94.934,Y 90.606,Z 83.945,A 180.000,B 0.000,C 180.000} C_DIS
LIN {X 94.797,Y 90.657,Z 83.942,A 180.000,B 0.000,C 180.000} C_DIS
LIN {X 94.663,Y 90.710,Z 83.939,A 180.000,B 0.000,C 180.000} C_DIS
LIN {X 94.531,Y 90.767,Z 83.936,A 180.000,B 0.000,C 180.000} C_DIS
LIN {X 94.389,Y 90.830,Z 83.932,A 180.000,B 0.000,C 180.000} C_DIS
LIN {X 94.249,Y 90.895,Z 83.929,A 180.000,B 0.000,C 180.000} C_DIS
LIN {X 94.119,Y 90.957,Z 83.925,A 180.000,B 0.000,C 180.000} C_DIS
LIN {X 93.990,Y 91.022,Z 83.922,A 180.000,B 0.000,C 180.000} C_DIS
LIN {X 93.857,Y 91.094,Z 83.918,A 180.000,B 0.000,C 180.000} C_DIS
LIN {X 93.727,Y 91.170,Z 83.914,A 180.000,B 0.000,C 180.000} C_DIS
LIN {X 93.598,Y 91.248,Z 83.910,A 180.000,B 0.000,C 180.000} C_DIS
LIN {X 93.471,Y 91.326,Z 83.906,A 180.000,B 0.000,C 180.000} C_DIS
LIN {X 93.343,Y 91.408,Z 83.902,A 180.000,B 0.000,C 180.000} C_DIS
LIN {X 93.216,Y 91.492,Z 83.898,A 180.000,B 0.000,C 180.000} C_DIS
LIN {X 93.098,Y 91.577,Z 83.894,A 180.000,B 0.000,C 180.000} C_DIS
LIN {X 92.981,Y 91.663,Z 83.890,A 180.000,B 0.000,C 180.000} C_DIS
LIN {X 92.865,Y 91.755,Z 83.885,A 180.000,B 0.000,C 180.000} C_DIS
LIN {X 92.750,Y 91.848,Z 83.881,A 180.000,B 0.000,C 180.000} C_DIS
LIN {X 92.636,Y 91.941,Z 83.877,A 180.000,B 0.000,C 180.000} C_DIS
LIN {X 92.523,Y 92.036,Z 83.872,A 180.000,B 0.000,C 180.000} C_DIS
LIN {X 92.414,Y 92.136,Z 83.868,A 180.000,B 0.000,C 180.000} C_DIS
LIN {X 92.306,Y 92.237,Z 83.863,A 180.000,B 0.000,C 180.000} C_DIS
LIN {X 92.198,Y 92.346,Z 83.858,A 180.000,B 0.000,C 180.000} C_DIS
LIN {X 92.091,Y 92.457,Z 83.854,A 180.000,B 0.000,C 180.000} C_DIS
LIN {X 91.985,Y 92.567,Z 83.849,A 180.000,B 0.000,C 180.000} C_DIS
LIN {X 91.881,Y 92.679,Z 83.844,A 180.000,B 0.000,C 180.000} C_DIS
LIN {X 91.788,Y 92.787,Z 83.839,A 180.000,B 0.000,C 180.000} C_DIS
LIN {X 91.696,Y 92.897,Z 83.834,A 180.000,B 0.000,C 180.000} C_DIS
LIN {X 91.649,Y 92.957,Z 83.832,A 180.000,B 0.000,C 180.000} C_DIS
LIN {X 91.602,Y 93.018,Z 83.829,A 180.000,B 0.000,C 180.000} C_DIS
LIN {X 91.555,Y 93.078,Z 83.827,A 180.000,B 0.000,C 180.000} C_DIS
LIN {X 91.509,Y 93.140,Z 83.824,A 180.000,B 0.000,C 180.000} C_DIS
LIN {X 91.419,Y 93.259,Z 83.819,A 180.000,B 0.000,C 180.000} C_DIS
LIN {X 91.375,Y 93.319,Z 83.816,A 180.000,B 0.000,C 180.000} C_DIS
LIN {X 91.333,Y 93.380,Z 83.814,A 180.000,B 0.000,C 180.000} C_DIS
LIN {X 91.291,Y 93.441,Z 83.811,A 180.000,B 0.000,C 180.000} C_DIS
LIN {X 91.248,Y 93.503,Z 83.808,A 180.000,B 0.000,C 180.000} C_DIS
LIN {X 91.207,Y 93.565,Z 83.806,A 180.000,B 0.000,C 180.000} C_DIS
LIN {X 91.168,Y 93.628,Z 83.803,A 180.000,B 0.000,C 180.000} C_DIS
LIN {X 91.090,Y 93.756,Z 83.798,A 180.000,B 0.000,C 180.000} C_DIS
LIN {X 91.052,Y 93.821,Z 83.795,A 180.000,B 0.000,C 180.000} C_DIS
LIN {X 91.015,Y 93.886,Z 83.793,A 180.000,B 0.000,C 180.000} C_DIS
LIN {X 90.939,Y 94.019,Z 83.787,A 180.000,B 0.000,C 180.000} C_DIS
LIN {X 90.902,Y 94.086,Z 83.785,A 180.000,B 0.000,C 180.000} C_DIS
LIN {X 90.865,Y 94.153,Z 83.782,A 180.000,B 0.000,C 180.000} C_DIS
LIN {X 90.831,Y 94.218,Z 83.780,A 180.000,B 0.000,C 180.000} C_DIS
LIN {X 90.796,Y 94.283,Z 83.777,A 180.000,B 0.000,C 180.000} C_DIS
LIN {X 90.764,Y 94.349,Z 83.774,A 180.000,B 0.000,C 180.000} C_DIS
LIN {X 90.733,Y 94.416,Z 83.772,A 180.000,B 0.000,C 180.000} C_DIS
LIN {X 90.701,Y 94.484,Z 83.769,A 180.000,B 0.000,C 180.000} C_DIS
LIN {X 90.670,Y 94.553,Z 83.767,A 180.000,B 0.000,C 180.000} C_DIS
LIN {X 90.640,Y 94.623,Z 83.764,A 180.000,B 0.000,C 180.000} C_DIS
LIN {X 90.611,Y 94.693,Z 83.761,A 180.000,B 0.000,C 180.000} C_DIS
LIN {X 90.552,Y 94.834,Z 83.756,A 180.000,B 0.000,C 180.000} C_DIS
LIN {X 90.523,Y 94.906,Z 83.753,A 180.000,B 0.000,C 180.000} C_DIS
LIN {X 90.495,Y 94.977,Z 83.751,A 180.000,B 0.000,C 180.000} C_DIS
LIN {X 90.468,Y 95.045,Z 83.748,A 180.000,B 0.000,C 180.000} C_DIS
LIN {X 90.442,Y 95.114,Z 83.745,A 180.000,B 0.000,C 180.000} C_DIS
LIN {X 90.419,Y 95.184,Z 83.743,A 180.000,B 0.000,C 180.000} C_DIS
LIN {X 90.395,Y 95.254,Z 83.740,A 180.000,B 0.000,C 180.000} C_DIS
LIN {X 90.371,Y 95.324,Z 83.738,A 180.000,B 0.000,C 180.000} C_DIS
LIN {X 90.349,Y 95.396,Z 83.735,A 180.000,B 0.000,C 180.000} C_DIS
LIN {X 90.329,Y 95.468,Z 83.732,A 180.000,B 0.000,C 180.000} C_DIS
LIN {X 90.309,Y 95.540,Z 83.730,A 180.000,B 0.000,C 180.000} C_DIS
LIN {X 90.288,Y 95.615,Z 83.727,A 180.000,B 0.000,C 180.000} C_DIS
LIN {X 90.247,Y 95.765,Z 83.722,A 180.000,B 0.000,C 180.000} C_DIS
LIN {X 90.226,Y 95.840,Z 83.719,A 180.000,B 0.000,C 180.000} C_DIS
LIN {X 90.208,Y 95.912,Z 83.716,A 180.000,B 0.000,C 180.000} C_DIS
LIN {X 90.192,Y 95.984,Z 83.714,A 180.000,B 0.000,C 180.000} C_DIS
LIN {X 90.160,Y 96.128,Z 83.709,A 180.000,B 0.000,C 180.000} C_DIS
LIN {X 90.145,Y 96.201,Z 83.706,A 180.000,B 0.000,C 180.000} C_DIS
LIN {X 90.133,Y 96.274,Z 83.703,A 180.000,B 0.000,C 180.000} C_DIS
LIN {X 90.109,Y 96.421,Z 83.698,A 180.000,B 0.000,C 180.000} C_DIS
LIN {X 90.098,Y 96.498,Z 83.696,A 180.000,B 0.000,C 180.000} C_DIS
LIN {X 90.076,Y 96.653,Z 83.690,A 180.000,B 0.000,C 180.000} C_DIS
LIN {X 90.064,Y 96.730,Z 83.687,A 180.000,B 0.000,C 180.000} C_DIS
LIN {X 90.055,Y 96.805,Z 83.685,A 180.000,B 0.000,C 180.000} C_DIS
LIN {X 90.048,Y 96.879,Z 83.682,A 180.000,B 0.000,C 180.000} C_DIS
LIN {X 90.040,Y 96.953,Z 83.680,A 180.000,B 0.000,C 180.000} C_DIS
LIN {X 90.033,Y 97.028,Z 83.677,A 180.000,B 0.000,C 180.000} C_DIS
LIN {X 90.027,Y 97.102,Z 83.674,A 180.000,B 0.000,C 180.000} C_DIS
LIN {X 90.024,Y 97.176,Z 83.672,A 180.000,B 0.000,C 180.000} C_DIS
LIN {X 90.021,Y 97.250,Z 83.669,A 180.000,B 0.000,C 180.000} C_DIS
LIN {X 90.017,Y 97.324,Z 83.667,A 180.000,B 0.000,C 180.000} C_DIS
LIN {X 90.015,Y 97.400,Z 83.664,A 180.000,B 0.000,C 180.000} C_DIS
LIN {X 90.013,Y 97.551,Z 83.659,A 180.000,B 0.000,C 180.000} C_DIS
LIN {X 90.012,Y 97.627,Z 83.656,A 180.000,B 0.000,C 180.000} C_DIS
LIN {X 90.012,Y 97.705,Z 83.653,A 180.000,B 0.000,C 180.000} C_DIS
LIN {X 90.014,Y 97.860,Z 83.648,A 180.000,B 0.000,C 180.000} C_DIS
LIN {X 90.016,Y 97.938,Z 83.645,A 180.000,B 0.000,C 180.000} C_DIS
LIN {X 90.020,Y 98.012,Z 83.642,A 180.000,B 0.000,C 180.000} C_DIS
LIN {X 90.030,Y 98.161,Z 83.637,A 180.000,B 0.000,C 180.000} C_DIS
LIN {X 90.036,Y 98.236,Z 83.635,A 180.000,B 0.000,C 180.000} C_DIS
LIN {X 90.044,Y 98.311,Z 83.632,A 180.000,B 0.000,C 180.000} C_DIS
LIN {X 90.060,Y 98.461,Z 83.627,A 180.000,B 0.000,C 180.000} C_DIS
LIN {X 90.069,Y 98.536,Z 83.624,A 180.000,B 0.000,C 180.000} C_DIS
LIN {X 90.078,Y 98.610,Z 83.622,A 180.000,B 0.000,C 180.000} C_DIS
LIN {X 90.087,Y 98.684,Z 83.619,A 180.000,B 0.000,C 180.000} C_DIS
LIN {X 90.096,Y 98.758,Z 83.616,A 180.000,B 0.000,C 180.000} C_DIS
LIN {X 90.108,Y 98.832,Z 83.614,A 180.000,B 0.000,C 180.000} C_DIS
LIN {X 90.121,Y 98.908,Z 83.611,A 180.000,B 0.000,C 180.000} C_DIS
LIN {X 90.135,Y 98.985,Z 83.608,A 180.000,B 0.000,C 180.000} C_DIS
LIN {X 90.149,Y 99.061,Z 83.606,A 180.000,B 0.000,C 180.000} C_DIS
LIN {X 90.165,Y 99.137,Z 83.603,A 180.000,B 0.000,C 180.000} C_DIS
LIN {X 90.182,Y 99.211,Z 83.600,A 180.000,B 0.000,C 180.000} C_DIS
LIN {X 90.218,Y 99.358,Z 83.595,A 180.000,B 0.000,C 180.000} C_DIS
LIN {X 90.235,Y 99.432,Z 83.592,A 180.000,B 0.000,C 180.000} C_DIS
LIN {X 90.271,Y 99.578,Z 83.587,A 180.000,B 0.000,C 180.000} C_DIS
LIN {X 90.289,Y 99.651,Z 83.584,A 180.000,B 0.000,C 180.000} C_DIS
LIN {X 90.310,Y 99.723,Z 83.582,A 180.000,B 0.000,C 180.000} C_DIS
LIN {X 90.354,Y 99.870,Z 83.576,A 180.000,B 0.000,C 180.000} C_DIS
LIN {X 90.377,Y 99.943,Z 83.574,A 180.000,B 0.000,C 180.000} C_DIS
LIN {X 90.402,Y 100.015,Z 83.571,A 180.000,B 0.000,C 180.000} C_DIS
LIN {X 90.454,Y 100.159,Z 83.566,A 180.000,B 0.000,C 180.000} C_DIS
LIN {X 90.481,Y 100.230,Z 83.563,A 180.000,B 0.000,C 180.000} C_DIS
LIN {X 90.535,Y 100.372,Z 83.558,A 180.000,B 0.000,C 180.000} C_DIS
LIN {X 90.561,Y 100.443,Z 83.555,A 180.000,B 0.000,C 180.000} C_DIS
LIN {X 90.590,Y 100.514,Z 83.552,A 180.000,B 0.000,C 180.000} C_DIS
LIN {X 90.619,Y 100.584,Z 83.550,A 180.000,B 0.000,C 180.000} C_DIS
LIN {X 90.649,Y 100.653,Z 83.547,A 180.000,B 0.000,C 180.000} C_DIS
LIN {X 90.679,Y 100.723,Z 83.545,A 180.000,B 0.000,C 180.000} C_DIS
LIN {X 90.711,Y 100.792,Z 83.542,A 180.000,B 0.000,C 180.000} C_DIS
LIN {X 90.745,Y 100.860,Z 83.539,A 180.000,B 0.000,C 180.000} C_DIS
LIN {X 90.779,Y 100.928,Z 83.537,A 180.000,B 0.000,C 180.000} C_DIS
LIN {X 90.813,Y 100.997,Z 83.534,A 180.000,B 0.000,C 180.000} C_DIS
LIN {X 90.848,Y 101.065,Z 83.531,A 180.000,B 0.000,C 180.000} C_DIS
LIN {X 90.920,Y 101.201,Z 83.526,A 180.000,B 0.000,C 180.000} C_DIS
LIN {X 90.956,Y 101.269,Z 83.523,A 180.000,B 0.000,C 180.000} C_DIS
LIN {X 90.994,Y 101.336,Z 83.520,A 180.000,B 0.000,C 180.000} C_DIS
LIN {X 91.069,Y 101.468,Z 83.515,A 180.000,B 0.000,C 180.000} C_DIS
LIN {X 91.107,Y 101.533,Z 83.513,A 180.000,B 0.000,C 180.000} C_DIS
LIN {X 91.147,Y 101.597,Z 83.510,A 180.000,B 0.000,C 180.000} C_DIS
LIN {X 91.230,Y 101.725,Z 83.505,A 180.000,B 0.000,C 180.000} C_DIS
LIN {X 91.272,Y 101.789,Z 83.502,A 180.000,B 0.000,C 180.000} C_DIS
LIN {X 91.316,Y 101.852,Z 83.499,A 180.000,B 0.000,C 180.000} C_DIS
LIN {X 91.404,Y 101.977,Z 83.494,A 180.000,B 0.000,C 180.000} C_DIS
LIN {X 91.448,Y 102.040,Z 83.491,A 180.000,B 0.000,C 180.000} C_DIS
LIN {X 91.538,Y 102.163,Z 83.486,A 180.000,B 0.000,C 180.000} C_DIS
LIN {X 91.583,Y 102.225,Z 83.483,A 180.000,B 0.000,C 180.000} C_DIS
LIN {X 91.630,Y 102.286,Z 83.480,A 180.000,B 0.000,C 180.000} C_DIS
LIN {X 91.679,Y 102.345,Z 83.478,A 180.000,B 0.000,C 180.000} C_DIS
LIN {X 91.727,Y 102.404,Z 83.475,A 180.000,B 0.000,C 180.000} C_DIS
LIN {X 91.775,Y 102.463,Z 83.472,A 180.000,B 0.000,C 180.000} C_DIS
LIN {X 91.825,Y 102.521,Z 83.470,A 180.000,B 0.000,C 180.000} C_DIS
LIN {X 91.876,Y 102.577,Z 83.467,A 180.000,B 0.000,C 180.000} C_DIS
LIN {X 91.979,Y 102.691,Z 83.462,A 180.000,B 0.000,C 180.000} C_DIS
LIN {X 92.031,Y 102.748,Z 83.459,A 180.000,B 0.000,C 180.000} C_DIS
LIN {X 92.084,Y 102.805,Z 83.456,A 180.000,B 0.000,C 180.000} C_DIS
LIN {X 92.136,Y 102.862,Z 83.454,A 180.000,B 0.000,C 180.000} C_DIS
LIN {X 92.189,Y 102.918,Z 83.451,A 180.000,B 0.000,C 180.000} C_DIS
LIN {X 92.244,Y 102.972,Z 83.448,A 180.000,B 0.000,C 180.000} C_DIS
LIN {X 92.353,Y 103.079,Z 83.443,A 180.000,B 0.000,C 180.000} C_DIS
LIN {X 92.408,Y 103.132,Z 83.440,A 180.000,B 0.000,C 180.000} C_DIS
LIN {X 92.465,Y 103.182,Z 83.438,A 180.000,B 0.000,C 180.000} C_DIS
LIN {X 92.579,Y 103.282,Z 83.432,A 180.000,B 0.000,C 180.000} C_DIS
LIN {X 92.638,Y 103.332,Z 83.430,A 180.000,B 0.000,C 180.000} C_DIS
LIN {X 92.756,Y 103.434,Z 83.424,A 180.000,B 0.000,C 180.000} C_DIS
LIN {X 92.815,Y 103.484,Z 83.422,A 180.000,B 0.000,C 180.000} C_DIS
LIN {X 92.875,Y 103.533,Z 83.419,A 180.000,B 0.000,C 180.000} C_DIS
LIN {X 92.997,Y 103.627,Z 83.413,A 180.000,B 0.000,C 180.000} C_DIS
LIN {X 93.058,Y 103.674,Z 83.411,A 180.000,B 0.000,C 180.000} C_DIS
LIN {X 93.119,Y 103.719,Z 83.408,A 180.000,B 0.000,C 180.000} C_DIS
LIN {X 93.181,Y 103.762,Z 83.405,A 180.000,B 0.000,C 180.000} C_DIS
LIN {X 93.244,Y 103.805,Z 83.403,A 180.000,B 0.000,C 180.000} C_DIS
LIN {X 93.306,Y 103.848,Z 83.400,A 180.000,B 0.000,C 180.000} C_DIS
LIN {X 93.371,Y 103.891,Z 83.397,A 180.000,B 0.000,C 180.000} C_DIS
LIN {X 93.501,Y 103.977,Z 83.392,A 180.000,B 0.000,C 180.000} C_DIS
LIN {X 93.566,Y 104.019,Z 83.389,A 180.000,B 0.000,C 180.000} C_DIS
LIN {X 93.631,Y 104.059,Z 83.387,A 180.000,B 0.000,C 180.000} C_DIS
LIN {X 93.760,Y 104.138,Z 83.381,A 180.000,B 0.000,C 180.000} C_DIS
LIN {X 93.826,Y 104.177,Z 83.379,A 180.000,B 0.000,C 180.000} C_DIS
LIN {X 93.894,Y 104.214,Z 83.376,A 180.000,B 0.000,C 180.000} C_DIS
LIN {X 94.031,Y 104.288,Z 83.371,A 180.000,B 0.000,C 180.000} C_DIS
LIN {X 94.100,Y 104.324,Z 83.368,A 180.000,B 0.000,C 180.000} C_DIS
LIN {X 94.168,Y 104.358,Z 83.365,A 180.000,B 0.000,C 180.000} C_DIS
LIN {X 94.306,Y 104.426,Z 83.360,A 180.000,B 0.000,C 180.000} C_DIS
LIN {X 94.376,Y 104.459,Z 83.357,A 180.000,B 0.000,C 180.000} C_DIS
LIN {X 94.514,Y 104.524,Z 83.352,A 180.000,B 0.000,C 180.000} C_DIS
LIN {X 94.584,Y 104.556,Z 83.349,A 180.000,B 0.000,C 180.000} C_DIS
LIN {X 94.654,Y 104.586,Z 83.346,A 180.000,B 0.000,C 180.000} C_DIS
LIN {X 94.726,Y 104.615,Z 83.344,A 180.000,B 0.000,C 180.000} C_DIS
LIN {X 94.798,Y 104.644,Z 83.341,A 180.000,B 0.000,C 180.000} C_DIS
LIN {X 94.871,Y 104.672,Z 83.338,A 180.000,B 0.000,C 180.000} C_DIS
LIN {X 94.944,Y 104.699,Z 83.336,A 180.000,B 0.000,C 180.000} C_DIS
LIN {X 95.017,Y 104.724,Z 83.333,A 180.000,B 0.000,C 180.000} C_DIS
LIN {X 95.163,Y 104.775,Z 83.327,A 180.000,B 0.000,C 180.000} C_DIS
LIN {X 95.237,Y 104.799,Z 83.325,A 180.000,B 0.000,C 180.000} C_DIS
LIN {X 95.309,Y 104.824,Z 83.322,A 180.000,B 0.000,C 180.000} C_DIS
LIN {X 95.382,Y 104.848,Z 83.319,A 180.000,B 0.000,C 180.000} C_DIS
LIN {X 95.455,Y 104.871,Z 83.317,A 180.000,B 0.000,C 180.000} C_DIS
LIN {X 95.529,Y 104.892,Z 83.314,A 180.000,B 0.000,C 180.000} C_DIS
LIN {X 95.679,Y 104.933,Z 83.309,A 180.000,B 0.000,C 180.000} C_DIS
LIN {X 95.754,Y 104.953,Z 83.306,A 180.000,B 0.000,C 180.000} C_DIS
LIN {X 95.829,Y 104.970,Z 83.303,A 180.000,B 0.000,C 180.000} C_DIS
LIN {X 95.981,Y 105.003,Z 83.298,A 180.000,B 0.000,C 180.000} C_DIS
LIN {X 96.057,Y 105.019,Z 83.295,A 180.000,B 0.000,C 180.000} C_DIS
LIN {X 96.133,Y 105.035,Z 83.292,A 180.000,B 0.000,C 180.000} C_DIS
LIN {X 96.209,Y 105.050,Z 83.290,A 180.000,B 0.000,C 180.000} C_DIS
LIN {X 96.285,Y 105.066,Z 83.287,A 180.000,B 0.000,C 180.000} C_DIS
LIN {X 96.361,Y 105.079,Z 83.284,A 180.000,B 0.000,C 180.000} C_DIS
LIN {X 96.437,Y 105.091,Z 83.282,A 180.000,B 0.000,C 180.000} C_DIS
LIN {X 96.513,Y 105.103,Z 83.279,A 180.000,B 0.000,C 180.000} C_DIS
LIN {X 96.589,Y 105.115,Z 83.276,A 180.000,B 0.000,C 180.000} C_DIS
LIN {X 96.665,Y 105.124,Z 83.274,A 180.000,B 0.000,C 180.000} C_DIS
LIN {X 96.742,Y 105.132,Z 83.271,A 180.000,B 0.000,C 180.000} C_DIS
LIN {X 96.820,Y 105.140,Z 83.268,A 180.000,B 0.000,C 180.000} C_DIS
LIN {X 96.897,Y 105.147,Z 83.265,A 180.000,B 0.000,C 180.000} C_DIS
LIN {X 96.975,Y 105.154,Z 83.263,A 180.000,B 0.000,C 180.000} C_DIS
LIN {X 97.053,Y 105.160,Z 83.260,A 180.000,B 0.000,C 180.000} C_DIS
LIN {X 97.131,Y 105.166,Z 83.257,A 180.000,B 0.000,C 180.000} C_DIS
LIN {X 97.208,Y 105.172,Z 83.254,A 180.000,B 0.000,C 180.000} C_DIS
LIN {X 97.286,Y 105.175,Z 83.252,A 180.000,B 0.000,C 180.000} C_DIS
LIN {X 97.364,Y 105.179,Z 83.249,A 180.000,B 0.000,C 180.000} C_DIS
LIN {X 97.441,Y 105.182,Z 83.246,A 180.000,B 0.000,C 180.000} C_DIS
LIN {X 97.518,Y 105.184,Z 83.244,A 180.000,B 0.000,C 180.000} C_DIS
LIN {X 97.595,Y 105.184,Z 83.241,A 180.000,B 0.000,C 180.000} C_DIS
LIN {X 97.672,Y 105.183,Z 83.238,A 180.000,B 0.000,C 180.000} C_DIS
LIN {X 97.750,Y 105.182,Z 83.236,A 180.000,B 0.000,C 180.000} C_DIS
LIN {X 97.827,Y 105.180,Z 83.233,A 180.000,B 0.000,C 180.000} C_DIS
LIN {X 97.905,Y 105.177,Z 83.230,A 180.000,B 0.000,C 180.000} C_DIS
LIN {X 97.983,Y 105.173,Z 83.227,A 180.000,B 0.000,C 180.000} C_DIS
LIN {X 98.061,Y 105.169,Z 83.225,A 180.000,B 0.000,C 180.000} C_DIS
LIN {X 98.139,Y 105.165,Z 83.222,A 180.000,B 0.000,C 180.000} C_DIS
LIN {X 98.296,Y 105.154,Z 83.217,A 180.000,B 0.000,C 180.000} C_DIS
LIN {X 98.373,Y 105.148,Z 83.214,A 180.000,B 0.000,C 180.000} C_DIS
LIN {X 98.450,Y 105.140,Z 83.211,A 180.000,B 0.000,C 180.000} C_DIS
LIN {X 98.526,Y 105.131,Z 83.208,A 180.000,B 0.000,C 180.000} C_DIS
LIN {X 98.603,Y 105.121,Z 83.206,A 180.000,B 0.000,C 180.000} C_DIS
LIN {X 98.680,Y 105.111,Z 83.203,A 180.000,B 0.000,C 180.000} C_DIS
LIN {X 98.757,Y 105.099,Z 83.200,A 180.000,B 0.000,C 180.000} C_DIS
LIN {X 98.833,Y 105.086,Z 83.198,A 180.000,B 0.000,C 180.000} C_DIS
LIN {X 98.987,Y 105.059,Z 83.192,A 180.000,B 0.000,C 180.000} C_DIS
LIN {X 99.063,Y 105.045,Z 83.189,A 180.000,B 0.000,C 180.000} C_DIS
LIN {X 99.140,Y 105.031,Z 83.187,A 180.000,B 0.000,C 180.000} C_DIS
LIN {X 99.216,Y 105.017,Z 83.184,A 180.000,B 0.000,C 180.000} C_DIS
LIN {X 99.293,Y 105.002,Z 83.181,A 180.000,B 0.000,C 180.000} C_DIS
LIN {X 99.369,Y 104.983,Z 83.179,A 180.000,B 0.000,C 180.000} C_DIS
LIN {X 99.445,Y 104.965,Z 83.176,A 180.000,B 0.000,C 180.000} C_DIS
LIN {X 99.521,Y 104.947,Z 83.173,A 180.000,B 0.000,C 180.000} C_DIS
LIN {X 99.597,Y 104.927,Z 83.171,A 180.000,B 0.000,C 180.000} C_DIS
LIN {X 99.671,Y 104.905,Z 83.168,A 180.000,B 0.000,C 180.000} C_DIS
LIN {X 99.745,Y 104.883,Z 83.166,A 180.000,B 0.000,C 180.000} C_DIS
LIN {X 99.820,Y 104.861,Z 83.163,A 180.000,B 0.000,C 180.000} C_DIS
LIN {X 99.894,Y 104.838,Z 83.161,A 180.000,B 0.000,C 180.000} C_DIS
LIN {X 99.969,Y 104.815,Z 83.158,A 180.000,B 0.000,C 180.000} C_DIS
LIN {X 100.043,Y 104.792,Z 83.156,A 180.000,B 0.000,C 180.000} C_DIS
LIN {X 100.118,Y 104.768,Z 83.153,A 180.000,B 0.000,C 180.000} C_DIS
LIN {X 100.192,Y 104.742,Z 83.151,A 180.000,B 0.000,C 180.000} C_DIS
LIN {X 100.266,Y 104.715,Z 83.148,A 180.000,B 0.000,C 180.000} C_DIS
LIN {X 100.413,Y 104.661,Z 83.143,A 180.000,B 0.000,C 180.000} C_DIS
LIN {X 100.556,Y 104.601,Z 83.138,A 180.000,B 0.000,C 180.000} C_DIS
LIN {X 100.700,Y 104.539,Z 83.134,A 180.000,B 0.000,C 180.000} C_DIS
LIN {X 100.842,Y 104.475,Z 83.129,A 180.000,B 0.000,C 180.000} C_DIS
LIN {X 100.984,Y 104.409,Z 83.124,A 180.000,B 0.000,C 180.000} C_DIS
LIN {X 101.124,Y 104.340,Z 83.120,A 180.000,B 0.000,C 180.000} C_DIS
LIN {X 101.263,Y 104.268,Z 83.115,A 180.000,B 0.000,C 180.000} C_DIS
LIN {X 101.399,Y 104.191,Z 83.111,A 180.000,B 0.000,C 180.000} C_DIS
LIN {X 101.534,Y 104.113,Z 83.106,A 180.000,B 0.000,C 180.000} C_DIS
LIN {X 101.667,Y 104.030,Z 83.102,A 180.000,B 0.000,C 180.000} C_DIS
LIN {X 101.801,Y 103.947,Z 83.098,A 180.000,B 0.000,C 180.000} C_DIS
LIN {X 101.932,Y 103.862,Z 83.094,A 180.000,B 0.000,C 180.000} C_DIS
LIN {X 102.060,Y 103.773,Z 83.089,A 180.000,B 0.000,C 180.000} C_DIS
LIN {X 102.187,Y 103.680,Z 83.085,A 180.000,B 0.000,C 180.000} C_DIS
LIN {X 102.311,Y 103.585,Z 83.081,A 180.000,B 0.000,C 180.000} C_DIS
LIN {X 102.434,Y 103.487,Z 83.078,A 180.000,B 0.000,C 180.000} C_DIS
LIN {X 102.555,Y 103.387,Z 83.074,A 180.000,B 0.000,C 180.000} C_DIS
LIN {X 102.676,Y 103.287,Z 83.070,A 180.000,B 0.000,C 180.000} C_DIS
LIN {X 102.793,Y 103.183,Z 83.067,A 180.000,B 0.000,C 180.000} C_DIS
LIN {X 102.908,Y 103.076,Z 83.063,A 180.000,B 0.000,C 180.000} C_DIS
LIN {X 103.019,Y 102.966,Z 83.060,A 180.000,B 0.000,C 180.000} C_DIS
LIN {X 103.128,Y 102.853,Z 83.056,A 180.000,B 0.000,C 180.000} C_DIS
LIN {X 103.237,Y 102.739,Z 83.053,A 180.000,B 0.000,C 180.000} C_DIS
LIN {X 103.345,Y 102.625,Z 83.050,A 180.000,B 0.000,C 180.000} C_DIS
LIN {X 103.448,Y 102.507,Z 83.047,A 180.000,B 0.000,C 180.000} C_DIS
LIN {X 103.550,Y 102.387,Z 83.044,A 180.000,B 0.000,C 180.000} C_DIS
LIN {X 103.647,Y 102.263,Z 83.041,A 180.000,B 0.000,C 180.000} C_DIS
